(* Logix 5000 project; controller QA_DC vendor 1 type 14 code 164 rev 32.16; software revision 32.04 *)

TASK MainTask (continuous, watchdog 500 ms) : MainProgram, LN99, LN98

MODULES
   Local : vendor 1 type 14 code 164 (ICP 2, rev 32.16)
      QA_DC_ETHERNET : 1756-EN2T (ICP 1, Ethernet 10.28.22.45, rev 11.1)
         Schedule_PreProd : vendor 1 type 14 code 236 (Ethernet 10.28.22.40, rev 31.1, $0ec75abb$ RPI 20 ms, $0e455032$ RPI 20 ms, $6b8e262d$ RPI 20 ms, $a9dcfd1c$ RPI 20 ms, $64bd79af$ RPI 20 ms, $7c715bd6$ RPI 20 ms, $9c0a19c1$ RPI 20 ms, $e338eee0$ RPI 20 ms, $88140ee3$ RPI 20 ms, $4102ecba$ RPI 20 ms, $cc31c595$ RPI 20 ms, $3449dfe4$ RPI 20 ms, $565c2e57$ RPI 20 ms, $e38346de$ RPI 20 ms, $e483dda9$ RPI 20 ms, $e8d43428$ RPI 20 ms, $2ed72c0b$ RPI 20 ms, $3992ee42$ RPI 20 ms, $82c155fd$ RPI 20 ms, $a33d8fac$ RPI 20 ms)
END_MODULES

TYPE Barcode_SNModel :
STRUCT
   Data : STRING[5];
   Bit : BOOL[32];
END_STRUCT
END_TYPE

TYPE DateTime :
STRUCT
   Year : DINT;
   Month : DINT;
   Day : DINT;
   Hour : DINT;
   Minute : DINT;
   Seconds : DINT;
   Microseconds : DINT;
END_STRUCT
END_TYPE

TYPE DateTime_Type :   // Structure for the DateTime from the Controller wallclock accessed by the GSV/SSV instruction
STRUCT
   Year : DINT;
   Month : DINT;   // The month (1 - 12)
   Day : DINT;   // The day (1 - 31)
   Hour : DINT;   // hour (0 - 23)
   Minute : DINT;   // minute (0 - 59)
   Second : DINT;   // second (0 - 59)
   Microseconds : DINT;   // (0 - 999,999)
END_STRUCT
END_TYPE

TYPE STRING_12 :
STRUCT
   LEN : DINT;
   DATA : SINT[12];
END_STRUCT
END_TYPE

TYPE STRING_16 :
STRUCT
   LEN : DINT;
   DATA : SINT[16];
END_STRUCT
END_TYPE

TYPE STRING_24 :
STRUCT
   LEN : DINT;
   DATA : SINT[24];
END_STRUCT
END_TYPE

TYPE STRING_4 :
STRUCT
   LEN : DINT;
   DATA : SINT[4];
END_STRUCT
END_TYPE

TYPE STRING_40 :
STRUCT
   LEN : DINT;
   DATA : SINT[40];
END_STRUCT
END_TYPE

TYPE UDT_Current_Status :
STRUCT
   Area : STRING_12;
   Line : STRING_12;
   Shift : DINT;
   _1st_Shift_Avail : BOOL;
   _1st_Shift_Active : BOOL;
   _1st_Shift_Scheduled : BOOL;
   _2nd_Shift_Avail : BOOL;
   _2nd_Shift_Active : BOOL;
   _2nd_Shift_Scheduled : BOOL;
   _3rd_Shift_Avail : BOOL;
   _3rd_Shift_Active : BOOL;
   _3rd_Shift_Scheduled : BOOL;
   DayOfWeek : STRING_16;
   DayOfWeek_Int : DINT;
   Start_Time : STRING_16;
   End_Time : STRING_16;
   _1st_Break_Time : STRING_16;
   _1st_Break_Trigger : BOOL;
   _1st_Break_Active : BOOL;
   _1st_Break_Used : BOOL;
   Lunch_Time : STRING_16;
   Lunch_Trigger : BOOL;
   Lunch_Active : BOOL;
   Lunch_Used : BOOL;
   _2nd_Break_Time : STRING_16;
   _2nd_Break_Trigger : BOOL;
   _2nd_Break_Active : BOOL;
   _2nd_Break_Used : BOOL;
   Rotate_Active : BOOL;
   Rotate_Cmd : BOOL;   // 30 Second Downtime Event to Rotate the Crew
   Scheduled_Units : DINT;
   Line_Rate : DINT;   // Seconds to Construct a Component
   Line_Rate_SP : REAL;
   Units_Remaining : DINT;
   Units_Produced : DINT;
   Units_Scrapped : DINT;
   Units_Lossed : DINT;
   AY_Percent : REAL;
   Shift_Minutes_Remainng : DINT;
   Shift_Seconds_Remaining : DINT;
   DownTime_Code : DINT;
   Flex_Cmd : BOOL;
   Flex_Active : BOOL;
   FlexTo_Line : STRING_16;
   Flex_EndCmd : BOOL;
   Rotate_LEN : REAL;   // seconds
   Brk_LEN : REAL;   // minutes
   Lunch_LEN : REAL;   // minutes
   Break_Stop_On : BOOL;
   Break_Stop_Allowed : BOOL;
   Flex_Stop_On : BOOL;
   Flex_Stop_Allowed : BOOL;
   Rotate_Stop_On : BOOL;
   Rotate_Stop_Allowed : BOOL;
   S1_Scheduled : DINT;
   S2_Scheduled : DINT;
   S3_Scheduled : DINT;
   Shift_Scheduled : BOOL;
   Shift_Active : BOOL;
   RateToMakeSchedule : REAL;
   Theoretical_Units : DINT;
   Standard_LineRate : REAL;
   Running : BOOL;
   State : DINT;
   LineWide_Event : DINT;
   Units_Rejected : DINT;
END_STRUCT
END_TYPE

TYPE UDT_Daily_Schedule :
STRUCT
   _1st_Shift_Avail : BOOL;
   _1st_Shift_Start : STRING_16;
   _1st_Shift_End : STRING_16;
   _1st_Shift_Break1_Start : STRING_16;
   _1st_Shift_Break1_Length : DINT;   // Minutes
   _1st_Shift_Lunch_Start : STRING_16;
   _1st_Shift_Lunch_Length : DINT;   // Minutes
   _1st_Shift_Break2_Start : STRING_16;
   _1st_Shift_Break2_Length : DINT;   // Minutes
   _2nd_Shift_Avail : BOOL;
   _2nd_Shift_Start : STRING_16;
   _2nd_Shift_End : STRING_16;
   _2nd_Shift_Break1_Start : STRING_16;
   _2nd_Shift_Break1_Length : DINT;   // Minutes
   _2nd_Shift_Lunch_Start : STRING_16;
   _2nd_Shift_Lunch_Length : DINT;   // Minutes
   _2nd_Shift_Break2_Start : STRING_16;
   _2nd_Shift_Break2_Length : DINT;   // Minutes
   _3rd_Shift_Avail : BOOL;
   _3rd_Shift_Start : STRING_16;
   _3rd_Shift_End : STRING_16;
   _3rd_Shift_Break1_Start : STRING_16;
   _3rd_Shift_Break1_Length : DINT;   // Minutes
   _3rd_Shift_Lunch_Start : STRING_16;
   _3rd_Shift_Lunch_Length : DINT;   // Minutes
   _3rd_Shift_Break2_Start : STRING_16;
   _3rd_Shift_Break2_Length : DINT;   // Minutes
   Rotate_Length : DINT;   // Seconds
   Break_Stop_On : BOOL;
   Break_Stop_Allowed : BOOL;
   Flex_Stop_On : BOOL;
   Flex_Stop_Allowed : BOOL;
   Rotate_Stop_On : BOOL;
   Rotate_Stop_Allowed : BOOL;
   S1_Scheduled : DINT;
   S2_Scheduled : DINT;
   S3_Scheduled : DINT;
   RateToMakeSchedule : REAL;
END_STRUCT
END_TYPE

TYPE UDT_ShiftString_Breakdown :
STRUCT
   s1StartHour : STRING_4;
   s1StartMin : STRING_4;
   s1EndHour : STRING_4;
   s1_EndMin : STRING_4;
   s2StartHour : STRING_4;
   s2StartMin : STRING_4;
   s2EndHour : STRING_4;
   s2EndMin : STRING_4;
   s3StartHour : STRING_4;
   s3StartMin : STRING_4;
   s3EndHour : STRING_4;
   s3EndMin : STRING_4;
   break1StartHour : STRING_4;
   break1StartMin : STRING_4;
   break2StartHour : STRING_4;
   break2StartMin : STRING_4;
   lunchStartHour : STRING_4;
   lunchStartMin : STRING_4;
END_STRUCT
END_TYPE

TYPE UDT_SN_Model :
STRUCT
   writeIndex : DINT;
   readIndex : DINT;
   LastReadCode : DINT;
   Serial : STRING_16;
   Model : STRING_16;
   DateTime : STRING_24;
   newData : BOOL;
END_STRUCT
END_TYPE

TYPE UDT_Weekly_Schedule :
STRUCT
   Monday : UDT_Daily_Schedule;
   Tuesday : UDT_Daily_Schedule;
   Wednesday : UDT_Daily_Schedule;
   Thursday : UDT_Daily_Schedule;
   Friday : UDT_Daily_Schedule;
   Saturday : UDT_Daily_Schedule;
   Sunday : UDT_Daily_Schedule;
END_STRUCT
END_TYPE

VAR_GLOBAL   (* controller tags *)
   LN98_1st_Station_Break_Code : DINT;
   LN98_Break_LineWide : BOOL := 1;
   LN98_Current_Shift_Duration_Mins : DINT;
   LN98_Current_Shift_Duration_wBreaks_Mins : DINT := 510;
   LN98_DC_Controlled_Theoretical_Units : BOOL := 1;
   LN98_DT_CODE : DINT;
   LN98_FROM_DC1_MAIN_MESSAGES : DINT[20] := ([3] := 1000); {produced}
   LN98_NewDataModelSerial : BOOL;
   LN98_PreviousSerialNumber : STRING := 'XA1018189';
   LN98_Schedule : UDT_Current_Status := (DayOfWeek_Int := 4, Units_Produced := 1020, Theoretical_Units := 1000, LineWide_Event := 16, Units_Rejected := 34);
   LN98_Schedule_Cycle_Timer : TIMER := (PRE := 30600, ACC := 30400);
   LN98_Schedule_Max_Break_Duration : DINT := 60;
   LN98_Schedule_Max_Break_Timer : TIMER := (PRE := 3600000, ACC := 3600000, DN := 1);
   LN98_Schedule_TAKT : REAL := 30600.0;
   LN98_Scheduled_Units_Buffer : DINT := 1000;
   LN98_SerialNumber_ONS : BOOL;
   LN98_SerialNumberBuffer : STRING;
   LN98_SerialNumberChange_DelayTimer : TIMER := (PRE := 2000);
   LN98_SerialNumberChange_Timer : TIMER := (PRE := 3000);
   LN98_Shift_Reset_ONS : BOOL;
   LN98_Theoretical_Units_Counter : COUNTER := (PRE := 999999, ACC := 999);
   LN98_Theoretical_Units_Counter_ONS : BOOL;
   LN98_TO_DC01_DOWNTIME_CODE : DINT[10];   // DOWNTIME CODE CONSUME TAG
        [0]   // LN98
        [1]   // WORK CENTER MAIN LINE A
        [2]   // WORK CENTER MAIN LINE B
        [3]   // WORK CENTER MAIN LINE C
        [4]   // WORK CENTER MAIN LINE D
        [5]   // WORK CENTER MAIN LINE E
        [6]   // WORK CENTER SUB LINE C
        [7]   // WORK CENTER SUB LINE E
   LN98_TO_DC01_MAIN_MESSAGES : DINT[20] := ([4] := 1020, [16] := 34);   // KPI CONSUME TAG
        [17]   // ACTIVE SHIFT
        [18]   // SCHEDULED UNITS
        [19]   // LOST UNIT COUNT
        [4]   // ACTUAL UNIT COUNT
        [9]   // LINE STATUS
        [9].0   // LINE RUNNING
        [9].1   // LINE ON BREAK
        [9].2   // LINE ON FLEX STOP
   LN98_TO_DC01_MODEL_SERIAL_MESSAGE : STRING[2] := ([0] := 'WAXXXXXXXX 19', [1] := 'XA1018189');
   LN98_TO_DC1_MAIN_MESSAGE_A : DINT[10];   // WORK CENTER A CONSUME TAG
   LN98_TO_DC1_MAIN_MESSAGE_B : DINT[10];   // WORK CENTER B CONSUME TAG
   LN98_TO_DC1_MAIN_MESSAGE_C : DINT[10];   // WORK CENTER C CONSUME TAG
   LN98_TO_DC1_MAIN_MESSAGE_D : DINT[10];   // WORK CENTER D CONSUME TAG
   LN98_TO_DC1_MAIN_MESSAGE_E : DINT[10];   // WORK CENTER E CONSUME TAG
   LN98_TO_DC1_SUB_MESSAGE_C : DINT[10];   // WORK CENTER C CONSUME TAG
   LN98_TO_DC1_SUB_MESSAGE_E : DINT[10];   // WORK CENTER E CONSUME TAG
   LN98_Weekly_Schedule : UDT_Weekly_Schedule := (Monday._1st_Shift_Avail := 1, Monday._1st_Shift_Start := '2023-05-22 05:00', Monday._1st_Shift_End := '2023-05-22 14:30', Monday._2nd_Shift_Avail := 1, Monday._2nd_Shift_Start := '2023-05-22 16:45', Monday._2nd_Shift_End := '2023-05-23 03:15', Monday._3rd_Shift_Start := '2023-05-22 04:50', Monday._3rd_Shift_End := '2023-05-22 04:55', Monday.S1_Scheduled := 1000, Monday.S2_Scheduled := 1000, Tuesday._1st_Shift_Avail := 1, Tuesday._1st_Shift_Start := '2023-05-23 05:00', Tuesday._1st_Shift_End := '2023-05-23 14:30', Tuesday._2nd_Shift_Avail := 1, Tuesday._2nd_Shift_Start := '2023-05-23 16:45', Tuesday._2nd_Shift_End := '2023-05-24 03:15', Tuesday._3rd_Shift_Start := '2023-05-23 04:50', Tuesday._3rd_Shift_End := '2023-05-23 04:55', Tuesday.S1_Scheduled := 1000, Tuesday.S2_Scheduled := 1000, Wednesday._1st_Shift_Avail := 1, Wednesday._1st_Shift_Start := '2023-05-24 05:00', Wednesday._1st_Shift_End := '2023-05-24 14:30', Wednesday._2nd_Shift_Avail := 1, Wednesday._2nd_Shift_Start := '2023-05-24 16:45', Wednesday._2nd_Shift_End := '2023-05-25 03:15', Wednesday._3rd_Shift_Start := '2023-05-24 04:50', Wednesday._3rd_Shift_End := '2023-05-24 04:55', Wednesday.S1_Scheduled := 1000, Wednesday.S2_Scheduled := 1000, Thursday._1st_Shift_Avail := 1, Thursday._1st_Shift_Start := '2023-05-18 05:00', Thursday._1st_Shift_End := '2023-05-18 14:30', Thursday._2nd_Shift_Avail := 1, Thursday._2nd_Shift_Start := '2023-05-18 16:45', Thursday._2nd_Shift_End := '2023-05-19 03:15', Thursday._3rd_Shift_Start := '2023-05-18 04:50', Thursday._3rd_Shift_End := '2023-05-18 04:55', Thursday.S1_Scheduled := 1000, Thursday.S2_Scheduled := 1000, Friday._1st_Shift_Avail := 1, Friday._1st_Shift_Start := '2023-05-19 05:00', Friday._1st_Shift_End := '2023-05-19 14:30', Friday._2nd_Shift_Avail := 1, Friday._2nd_Shift_Start := '2023-05-19 16:45', Friday._2nd_Shift_End := '2023-05-20 03:15', Friday._3rd_Shift_Start := '2023-05-19 04:50', Friday._3rd_Shift_End := '2023-05-19 04:55', Friday.S1_Scheduled := 1000, Friday.S2_Scheduled := 1000, Saturday._1st_Shift_Start := '2023-05-20 05:00', Saturday._1st_Shift_End := '2023-05-20 14:30', Saturday._2nd_Shift_Start := '2023-05-20 16:45', Saturday._2nd_Shift_End := '2023-05-21 01:15', Saturday._3rd_Shift_Start := '2023-05-20 04:50', Saturday._3rd_Shift_End := '2023-05-20 04:55', Sunday._1st_Shift_Start := '2023-05-21 05:00', Sunday._1st_Shift_End := '2023-05-21 14:30', Sunday._2nd_Shift_Start := '2023-05-21 16:45', Sunday._2nd_Shift_End := '2023-05-22 01:15',
        Sunday._3rd_Shift_Start := '2023-05-21 04:50', Sunday._3rd_Shift_End := '2023-05-21 04:55');
   LN98_WORKCENTER_MAINLINE_A_DT_CODE : DINT;
   LN98_WORKCENTER_MAINLINE_B_DT_CODE : DINT;
   LN98_WORKCENTER_MAINLINE_C_DT_CODE : DINT;
   LN98_WORKCENTER_MAINLINE_D_DT_CODE : DINT;
   LN98_WORKCENTER_MAINLINE_E_DT_CODE : DINT;
   LN98_WORKCENTER_SUBLINE_C_DT_CODE : DINT;
   LN98_WORKCENTER_SUBLINE_E_DT_CODE : DINT;
   LN98ECS01 : DINT;
   LN98ECS02 : DINT;
   LN98ECS03 : DINT;
   LN98EES01 : DINT;
   LN98EES02 : DINT;
   LN98EES03 : DINT;
   LN98NAM01 : DINT;
   LN98NAM02 : DINT;
   LN98NAM03 : DINT;
   LN98NAM04 : DINT;
   LN98NBM01 : DINT;
   LN98NBM02 : DINT;
   LN98NBM03 : DINT;
   LN98NBM04 : DINT;
   LN98NCM01 : DINT;
   LN98NCM02 : DINT;
   LN98NCM04 : DINT;
   LN98NCM05 : DINT;
   LN98NDM01 : DINT;
   LN98NDM02 : DINT;
   LN98NDM03 : DINT;
   LN98NDM04 : DINT;
   LN98NEM01 : DINT;
   LN98NEM02 : DINT;
   LN98NEM03 : DINT;
   LN98NEM04 : DINT;
   LN98NEM05 : DINT;
   LN98SAM01 : DINT;
   LN98SAM02 : DINT;
   LN98SAM03 : DINT;
   LN98SAM04 : DINT;
   LN98SBM01 : DINT;
   LN98SBM02 : DINT;
   LN98SBM03 : DINT;
   LN98SBM04 : DINT;
   LN98SCM01 : DINT;
   LN98SCM02 : DINT;
   LN98SCM03 : DINT;
   LN98SCM04 : DINT;
   LN98SCM05 : DINT;
   LN98SDM01 : DINT;
   LN98SDM02 : DINT;
   LN98SDM03 : DINT;
   LN98SDM04 : DINT;
   LN98SEM01 : DINT;
   LN98SEM02 : DINT;
   LN98SEM04 : DINT;
   LN98SEM05 : DINT;
   LN98WCS01 : DINT;
   LN98WCS02 : DINT;
   LN98WCS03 : DINT;
   LN98WES01 : DINT;
   LN98WES02 : DINT;
   LN98WES03 : DINT;
   LN99_1st_Station_Break_Code : DINT;
   LN99_Break_LineWide : BOOL := 1;
   LN99_Current_Shift_Duration_Mins : DINT;
   LN99_Current_Shift_Duration_wBreaks_Mins : DINT := 460;
   LN99_DC_Controlled_Theoretical_Units : BOOL := 1;
   LN99_DT_CODE : DINT;
   LN99_FROM_DC1_MAIN_MESSAGES : DINT[20] := ([3] := 600); {produced}
   LN99_NewDataModelSerial : BOOL;
   LN99_PreviousSerialNumber : STRING := 'XB1017079';
   LN99_Schedule : UDT_Current_Status := (Line := 'LN01', _1st_Shift_Scheduled := 1, _2nd_Shift_Scheduled := 1, DayOfWeek := 'Tue', DayOfWeek_Int := 4, Start_Time := '2023-03-23 05:00', End_Time := '2023-03-23 14:30', Units_Remaining := 1452, Units_Produced := 766, Units_Lossed := 65, AY_Percent := 95.02853, Theoretical_Units := 1240, LineWide_Event := 16, Units_Rejected := 38);
   LN99_Schedule_Cycle_Timer : TIMER := (PRE := 22258, ACC := 2761);
   LN99_Schedule_Max_Break_Duration : DINT := 50;
   LN99_Schedule_Max_Break_Timer : TIMER := (PRE := 3000000, ACC := 2999998);
   LN99_Schedule_TAKT : REAL := 22258.064;
   LN99_Scheduled_Units_Buffer : DINT := 1240;
   LN99_SerialNumber_ONS : BOOL;
   LN99_SerialNumberBuffer : STRING;
   LN99_SerialNumberChange_DelayTimer : TIMER := (PRE := 2000);
   LN99_SerialNumberChange_Timer : TIMER := (PRE := 3000);
   LN99_Shift_Reset_ONS : BOOL;
   LN99_Theoretical_Units_Counter : COUNTER := (PRE := 999999, ACC := 1240);
   LN99_Theoretical_Units_Counter_ONS : BOOL;
   LN99_TO_DC01_DOWNTIME_CODE : DINT[10];   // DOWNTIME CODE CONSUME TAG
        [0]   // LN 99
        [1]   // WORK CENTER MAIN LINE A
        [2]   // WORK CENTER MAIN LINE B
        [3]   // WORK CENTER MAIN LINE C
        [4]   // WORK CENTER MAIN LINE D
        [5]   // WORK CENTER MAIN LINE E
        [6]   // WORK CENTER SUB LINE C
        [7]   // WORK CENTER SUB LINE E
   LN99_TO_DC01_MAIN_MESSAGES : DINT[20] := ([4] := 766, [16] := 38);   // KPI CONSUME TAG
        [17]   // ACTIVE SHIFT
        [18]   // SCHEDULED UNITS
        [19]   // LOST UNIT COUNT
        [4]   // ACTUAL UNIT COUNT
        [9]   // LINE STATUS
        [9].0   // LINE RUNNING
        [9].1   // LINE ON BREAK
        [9].2   // LINE ON FLEX STOP
   LN99_TO_DC01_MODEL_SERIAL_MESSAGE : STRING[2] := ([0] := 'WBXXXXXXXX 13', [1] := 'XB1017079');
   LN99_TO_DC1_MAIN_MESSAGE_A : DINT[10];   // WORK CENTER A CONSUME TAG
        [1]   // LN99NAM01
        [2]   // LN99SAM01
        [3]   // LN99NAM02
        [4]   // LN99SAM02
        [5]   // LN99NAM03
        [6]   // LN99SAM03
        [7]   // LN99NAM04
        [8]   // LN99SAM04
   LN99_TO_DC1_MAIN_MESSAGE_B : DINT[10];   // WORK CENTER B CONSUME TAG
        [1]   // LN99NBM01 WORK STATION
        [2]   // LN99SBM01 WORK STATION
        [3]   // LN99NBM02 WORK STATION
        [4]   // LN99SBM02 WORK STATION
        [5]   // LN99NBM03 WORK STATION
        [6]   // LN99SBM03 WORK STATION
        [7]   // LN99NBM04 WORK STATION
        [8]   // LN99SBM04 WORK STATION
   LN99_TO_DC1_MAIN_MESSAGE_C : DINT[10];   // WORK CENTER C CONSUME TAG
        [1]   // LN99NCM01 WORK STATION
        [2]   // LN99SCM01 WORK STATION
        [3]   // LN99NCM02 WORK STATION
        [4]   // LN99SCM02 WORK STATION
        [5]   // LN99SCM03 WORK STATION
        [6]   // LN99NCM04 WORK STATION
        [7]   // LN99SCM04 WORK STATION
        [8]   // LN99NCM05 WORK STATION
        [9]   // LN99SCM05 WORK STATION
   LN99_TO_DC1_MAIN_MESSAGE_D : DINT[10];   // WORK CENTER D CONSUME TAG
        [1]   // LN99NDM01 WORK STATION
        [2]   // LN99SDM01 WORK STATION
        [3]   // LN99NDM02 WORK STATION
        [4]   // LN99SDM02 WORK STATION
        [5]   // LN99NDM03 WORK STATION
        [6]   // LN99SDM03 WORK STATION
        [7]   // LN99NDM04 WORK STATION
        [8]   // LN99SDM04 WORK STATION
   LN99_TO_DC1_MAIN_MESSAGE_E : DINT[10];   // WORK CENTER E CONSUME TAG
        [1]   // LN99NEM01 WORK STATION
        [2]   // LN99SEM01 WORK STATION
        [3]   // LN99NEM02 WORK STATION
        [4]   // LN99SEM02 WORK STATION
        [5]   // LN99NEM03 WORK STATION
        [6]   // LN99NEM04 WORK STATION
        [7]   // LN99SEM04 WORK STATION
        [8]   // LN99NEM05 WORK STATION
        [9]   // LN99SEM05 WORK STATION
   LN99_TO_DC1_SUB_MESSAGE_C : DINT[10];   // WORK CENTER C CONSUME TAG
        [1]   // LN99WCS01 WORK STATION
        [2]   // LN99ECS01 WORK STATION
        [3]   // LN99WCS02 WORK STATION
        [4]   // LN99ECS02 WORK STATION
        [5]   // LN99WCS03 WORK STATION
        [6]   // LN99ECS03 WORK STATION
   LN99_TO_DC1_SUB_MESSAGE_E : DINT[10];   // WORK CENTER E CONSUME TAG
        [1]   // LN99WES01 WORK STATION
        [2]   // LN99EES01 WORK STATION
        [3]   // LN99WES02 WORK STATION
        [4]   // LN99EES02 WORK STATION
        [5]   // LN99WES03 WORK STATION
        [6]   // LN99EES03 WORK STATION
   LN99_Weekly_Schedule : UDT_Weekly_Schedule := (Monday._1st_Shift_Avail := 1, Monday._1st_Shift_Start := '2023-05-22 05:00', Monday._1st_Shift_End := '2023-05-22 13:30', Monday._2nd_Shift_Avail := 1, Monday._2nd_Shift_Start := '2023-05-22 16:45', Monday._2nd_Shift_End := '2023-05-23 01:15', Monday._3rd_Shift_Start := '2023-05-22 04:50', Monday._3rd_Shift_End := '2023-05-22 04:55', Monday.S1_Scheduled := 1240, Monday.S2_Scheduled := 1240, Tuesday._1st_Shift_Avail := 1, Tuesday._1st_Shift_Start := '2023-05-23 05:00', Tuesday._1st_Shift_End := '2023-05-23 13:30', Tuesday._2nd_Shift_Avail := 1, Tuesday._2nd_Shift_Start := '2023-05-23 16:45', Tuesday._2nd_Shift_End := '2023-05-24 01:15', Tuesday._3rd_Shift_Start := '2023-05-23 04:50', Tuesday._3rd_Shift_End := '2023-05-23 04:55', Tuesday.S1_Scheduled := 1240, Tuesday.S2_Scheduled := 1240, Wednesday._1st_Shift_Avail := 1, Wednesday._1st_Shift_Start := '2023-05-24 05:00', Wednesday._1st_Shift_End := '2023-05-24 13:30', Wednesday._2nd_Shift_Avail := 1, Wednesday._2nd_Shift_Start := '2023-05-24 16:45', Wednesday._2nd_Shift_End := '2023-05-25 01:15', Wednesday._3rd_Shift_Start := '2023-05-24 04:50', Wednesday._3rd_Shift_End := '2023-05-24 04:55', Wednesday.S1_Scheduled := 1240, Wednesday.S2_Scheduled := 1240, Thursday._1st_Shift_Avail := 1, Thursday._1st_Shift_Start := '2023-05-18 05:00', Thursday._1st_Shift_End := '2023-05-18 13:30', Thursday._2nd_Shift_Avail := 1, Thursday._2nd_Shift_Start := '2023-05-18 16:45', Thursday._2nd_Shift_End := '2023-05-19 01:15', Thursday._3rd_Shift_Start := '2023-05-18 04:50', Thursday._3rd_Shift_End := '2023-05-18 04:55', Thursday.S1_Scheduled := 1240, Thursday.S2_Scheduled := 1240, Friday._1st_Shift_Avail := 1, Friday._1st_Shift_Start := '2023-05-19 05:00', Friday._1st_Shift_End := '2023-05-19 13:30', Friday._2nd_Shift_Avail := 1, Friday._2nd_Shift_Start := '2023-05-19 16:45', Friday._2nd_Shift_End := '2023-05-20 01:15', Friday._3rd_Shift_Start := '2023-05-19 04:50', Friday._3rd_Shift_End := '2023-05-19 04:55', Friday.S1_Scheduled := 1240, Friday.S2_Scheduled := 1240, Saturday._1st_Shift_Start := '2023-05-20 05:00', Saturday._1st_Shift_End := '2023-05-20 13:30', Saturday._2nd_Shift_Start := '2023-05-20 16:45', Saturday._2nd_Shift_End := '2023-05-21 01:15', Saturday._3rd_Shift_Start := '2023-05-20 04:50', Saturday._3rd_Shift_End := '2023-05-20 04:55', Saturday.S1_Scheduled := 1240, Saturday.S2_Scheduled := 1240, Sunday._1st_Shift_Start := '2023-05-21 05:00', Sunday._1st_Shift_End := '2023-05-21 13:30',
        Sunday._2nd_Shift_Start := '2023-05-21 16:45', Sunday._2nd_Shift_End := '2023-05-22 01:15', Sunday._3rd_Shift_Start := '2023-05-21 04:50', Sunday._3rd_Shift_End := '2023-05-21 04:55', Sunday.S1_Scheduled := 1240, Sunday.S2_Scheduled := 1240);
   LN99_WORKCENTER_MAINLINE_A_DT_CODE : DINT;
   LN99_WORKCENTER_MAINLINE_B_DT_CODE : DINT;
   LN99_WORKCENTER_MAINLINE_C_DT_CODE : DINT;
   LN99_WORKCENTER_MAINLINE_D_DT_CODE : DINT;
   LN99_WORKCENTER_MAINLINE_E_DT_CODE : DINT;
   LN99_WORKCENTER_SUBLINE_C_DT_CODE : DINT;
   LN99_WORKCENTER_SUBLINE_E_DT_CODE : DINT;
   LN99ECS01 : DINT;   // WORK STATION EAST SIDE WORKCENTER C SUBLINE STATION 01
   LN99ECS02 : DINT;   // WORK STATION EAST SIDE WORKCENTER C SUBLINE STATION 02
   LN99ECS03 : DINT;   // WORK STATION EAST SIDE WORKCENTER C SUBLINE STATION 03
   LN99EES01 : DINT;   // WORK STATION EAST SIDE WORK CENTER E SUBLINE STATION 01
   LN99EES02 : DINT;   // WORK STATION EAST SIDE WORK CENTER E SUBLINE STATION 02
   LN99EES03 : DINT;   // WORK STATION EAST SIDE WORK CENTER E SUBLINE STATION 03
   LN99NAM01 : DINT;   // WORKSTATION NORTH SIDE WORKCENTER A MAIN LINE STATION 01
   LN99NAM02 : DINT;   // WORKSTATION NORTH SIDE WORKCENTER A MAINLINE STATION 02
   LN99NAM03 : DINT;   // WORKSTATION NORTH SIDE WORKCENTER A MAINLINE STATION 03
   LN99NAM04 : DINT;   // WORKSTATION NORTH SIDE WORKCENTER A MAINLINE STATION 04
   LN99NBM01 : DINT;   // WORK STATION NORTH SIDE WORKCENTER B MAINLINE STATION 01
   LN99NBM02 : DINT;   // WORK STATION NORTH SIDE WORKCENTER B MAINLINE STATION 02
   LN99NBM03 : DINT;   // WORK STATION NORTH SIDE WORKCENTER B MAINLINE STATION 03
   LN99NBM04 : DINT;   // WORK STATION NORTH SIDE WORKCENTER B MAINLINE STATION 4
   LN99NCM01 : DINT;   // WORK STATION NORTH SIDE WORKCENTER C MAINLINE STATION 01
   LN99NCM02 : DINT;   // WORK STATION NORTH SIDE WORKCENTER C MAINLINE STATION 02
   LN99NCM04 : DINT;   // WORK STATION NORTH SIDE WORKCENTER C MAINLINE STATION 04
   LN99NCM05 : DINT;   // WORK STATION NORTH SIDE WORKCENTER C MAINLINE STATION 05
   LN99NDM01 : DINT;   // WORK STATION NORTH SIDE WORKCENTER D MAINLINE STATION 01
   LN99NDM02 : DINT;   // WORK STATION NORTH SIDE WORK CENTER D MAINLINE STATION 02
   LN99NDM03 : DINT;   // WORK STATION NORTH SIDE WORK CENTER D MAINLINE STATION 03
   LN99NDM04 : DINT;   // WORK STATION NORTH SIDE WORK CENTER D MAINLINE STATION 04
   LN99NEM01 : DINT;   // WORK STATION NORTH SIDE WORK CENTER E MAIN LINE STATION 01
   LN99NEM02 : DINT;   // WORK STATION NORTH SIDE WORK CENTER E MAINLINE STATION 02
   LN99NEM03 : DINT;   // WORK STATION NORTH SIDE WORK CENTER E MAINLINE STATION 03
   LN99NEM04 : DINT;   // WORK STATION NORTH SIDE WORK CENTER E MAINLINE STATION 04
   LN99NEM05 : DINT;   // WORK STATION NORTH SIDE WORK CENTER E MAINLINE STATION 05
   LN99SAM01 : DINT;   // WORKSTATION SOUTH SIDE WORKCENTER A MAIN LINE STATION 01
   LN99SAM02 : DINT;   // WORKSTATION SOUTH SIDE WORKCENTER A MAINLINE STATION 02
   LN99SAM03 : DINT;   // WORKSTATION SOUTH SIDE WORKCENTER A MAINLINE STATION 03
   LN99SAM04 : DINT;   // WORKSTATION SOUTH SIDE WORKCENTER A MAINLINE STATION 04
   LN99SBM01 : DINT;   // WORK STATION SOUTH SIDE WORKCENTER B MAINLINE STATION 01
   LN99SBM02 : DINT;   // WORK STATION SOUTH SIDE WORKCENTER B MAINLINE STATION 02
   LN99SBM03 : DINT;   // WORK STATION SOUTH SIDE WORKCENTER B MAINLINE STATION 03
   LN99SBM04 : DINT;   // WORK STATION SOUTH SIDE WORKCENTER B MAINLINE STATION 04
   LN99SCM01 : DINT;   // WORK STATION SOUTH SIDE WORKCENTER C MAINLINE STATION 01
   LN99SCM02 : DINT;   // WORK STATION SOUTH SIDE WORKCENTER C MAINLINE STATION 02
   LN99SCM03 : DINT;   // WORK STATION SOUTH SIDE WORKCENTER C MAINLINE STATION 03
   LN99SCM04 : DINT;   // WORK STATION SOUTH SIDE WORKCENTER C MAINLINE STATION 04
   LN99SCM05 : DINT;   // WORK STATION SOUTH SIDE WORKCENTER C MAINLINE STATION 05
   LN99SDM01 : DINT;   // WORK STATION SOUTH SIDE WORKCENTER D MAINLINE STATION 01
   LN99SDM02 : DINT;   // WORK STATION SOUTH SIDE WORK CENTER D MAINLINE STATION 02
   LN99SDM03 : DINT;   // WORK STATION SOUTH SIDE WORK CENTER D MAINLINE STATION 03
   LN99SDM04 : DINT;   // WORK STATION SOUTH SIDE WORK CENTER D MAINLINE STATION 04
   LN99SEM01 : DINT;   // WORK STATION SOUTH SIDE WORK CENTER E MAINLINE STATION 01
   LN99SEM02 : DINT;   // WORK STATION SOUTH SIDE WORK CENTER E MAINLINE STATION 02
   LN99SEM04 : DINT;   // WORK STATION SOUTH SIDE WORK CENTER E MAINLINE STATION 04
   LN99SEM05 : DINT;   // WORK STATION SOUTH SIDE WORK CENTER E MAINLINE STATION 05
   LN99WCS01 : DINT;   // WORK STATION WEST SIDE WORKCENTER C SUBLINE STATION 01
   LN99WCS02 : DINT;   // WORK STATION WEST SIDE WORKCENTER C SUBLINE STATION 02
   LN99WCS03 : DINT;   // WORK STATION WEST SIDE WORKCENTER C SUBLINE STATION 03
   LN99WES01 : DINT;   // WORK STATION WEST SIDE WORK CENTER E SUBLINE STATION 01
   LN99WES02 : DINT;   // WORK STATION WEST SIDE WORK CENTER E SUBLINE STATION 02
   LN99WES03 : DINT;   // WORK STATION WEST SIDE WORK CENTER E SUBLINE STATION 03
END_VAR

PROGRAM LN98   (* main routine MainRoutine *)

ROUTINE MainRoutine   (* ladder *)
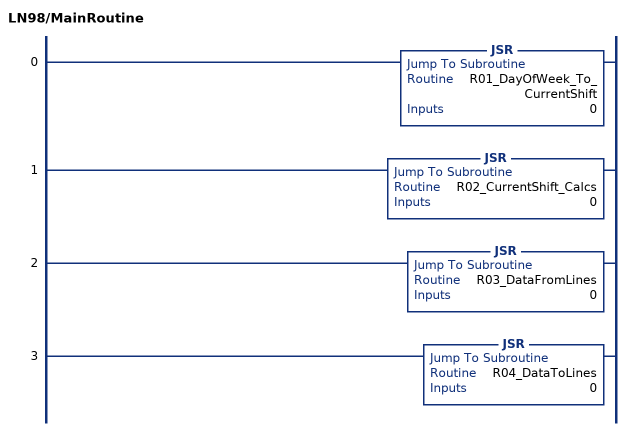
   0: JSR(R01_DayOfWeek_To_CurrentShift,0);
   1: JSR(R02_CurrentShift_Calcs,0);
   2: JSR(R03_DataFromLines,0);
   3: JSR(R04_DataToLines,0);
END_ROUTINE

ROUTINE R01_DayOfWeek_To_CurrentShift   (* ladder *)
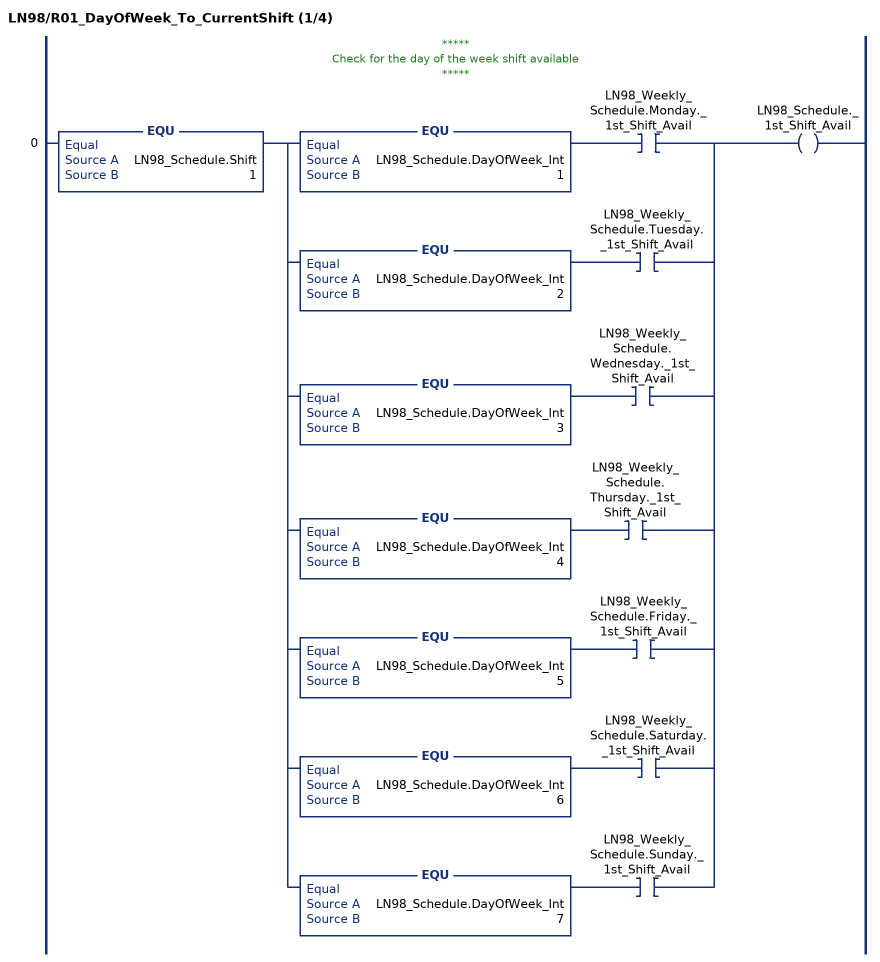
   // *****
   // Check for the day of the week shift available
   // *****
   0: EQU(LN98_Schedule.Shift,1)[EQU(LN98_Schedule.DayOfWeek_Int,1) XIC(LN98_Weekly_Schedule.Monday._1st_Shift_Avail) ,EQU(LN98_Schedule.DayOfWeek_Int,2) XIC(LN98_Weekly_Schedule.Tuesday._1st_Shift_Avail) ,EQU(LN98_Schedule.DayOfWeek_Int,3) XIC(LN98_Weekly_Schedule.Wednesday._1st_Shift_Avail) ,EQU(LN98_Schedule.DayOfWeek_Int,4) XIC(LN98_Weekly_Schedule.Thursday._1st_Shift_Avail) ,EQU(LN98_Schedule.DayOfWeek_Int,5) XIC(LN98_Weekly_Schedule.Friday._1st_Shift_Avail) ,EQU(LN98_Schedule.DayOfWeek_Int,6) XIC(LN98_Weekly_Schedule.Saturday._1st_Shift_Avail) ,EQU(LN98_Schedule.DayOfWeek_Int,7) XIC(LN98_Weekly_Schedule.Sunday._1st_Shift_Avail) ]OTE(LN98_Schedule._1st_Shift_Avail);
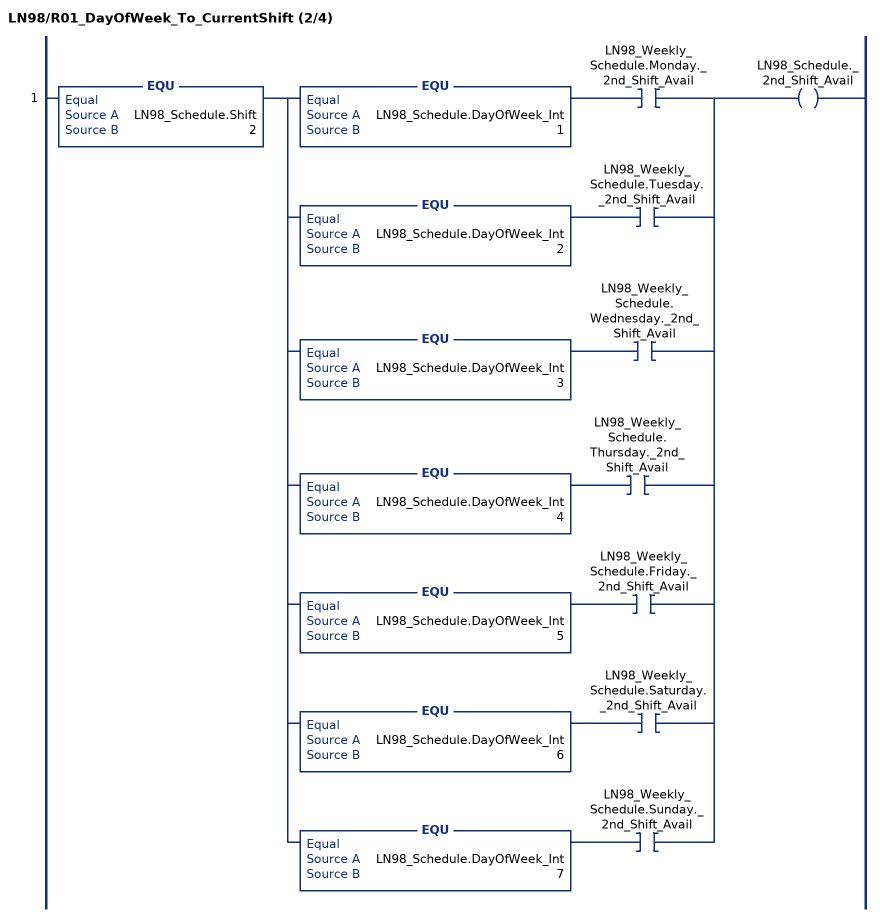
   1: EQU(LN98_Schedule.Shift,2)[EQU(LN98_Schedule.DayOfWeek_Int,1) XIC(LN98_Weekly_Schedule.Monday._2nd_Shift_Avail) ,EQU(LN98_Schedule.DayOfWeek_Int,2) XIC(LN98_Weekly_Schedule.Tuesday._2nd_Shift_Avail) ,EQU(LN98_Schedule.DayOfWeek_Int,3) XIC(LN98_Weekly_Schedule.Wednesday._2nd_Shift_Avail) ,EQU(LN98_Schedule.DayOfWeek_Int,4) XIC(LN98_Weekly_Schedule.Thursday._2nd_Shift_Avail) ,EQU(LN98_Schedule.DayOfWeek_Int,5) XIC(LN98_Weekly_Schedule.Friday._2nd_Shift_Avail) ,EQU(LN98_Schedule.DayOfWeek_Int,6) XIC(LN98_Weekly_Schedule.Saturday._2nd_Shift_Avail) ,EQU(LN98_Schedule.DayOfWeek_Int,7) XIC(LN98_Weekly_Schedule.Sunday._2nd_Shift_Avail) ]OTE(LN98_Schedule._2nd_Shift_Avail);
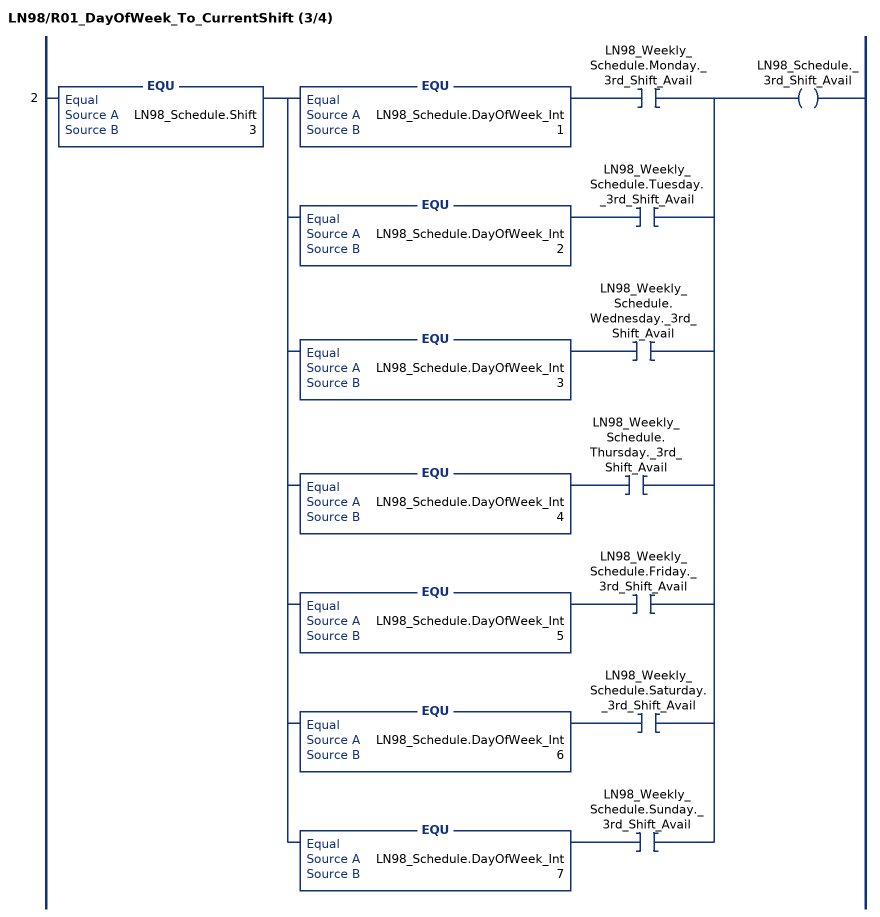
   2: EQU(LN98_Schedule.Shift,3)[EQU(LN98_Schedule.DayOfWeek_Int,1) XIC(LN98_Weekly_Schedule.Monday._3rd_Shift_Avail) ,EQU(LN98_Schedule.DayOfWeek_Int,2) XIC(LN98_Weekly_Schedule.Tuesday._3rd_Shift_Avail) ,EQU(LN98_Schedule.DayOfWeek_Int,3) XIC(LN98_Weekly_Schedule.Wednesday._3rd_Shift_Avail) ,EQU(LN98_Schedule.DayOfWeek_Int,4) XIC(LN98_Weekly_Schedule.Thursday._3rd_Shift_Avail) ,EQU(LN98_Schedule.DayOfWeek_Int,5) XIC(LN98_Weekly_Schedule.Friday._3rd_Shift_Avail) ,EQU(LN98_Schedule.DayOfWeek_Int,6) XIC(LN98_Weekly_Schedule.Saturday._3rd_Shift_Avail) ,EQU(LN98_Schedule.DayOfWeek_Int,7) XIC(LN98_Weekly_Schedule.Sunday._3rd_Shift_Avail) ]OTE(LN98_Schedule._3rd_Shift_Avail);
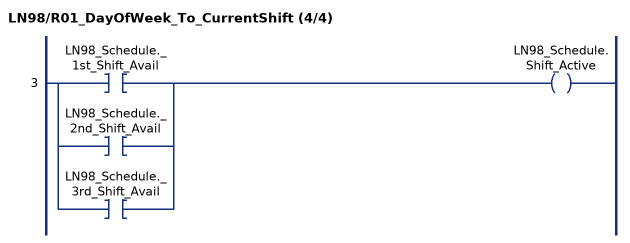
   3: [XIC(LN98_Schedule._1st_Shift_Avail) ,XIC(LN98_Schedule._2nd_Shift_Avail) ,XIC(LN98_Schedule._3rd_Shift_Avail) ]OTE(LN98_Schedule.Shift_Active);
END_ROUTINE

ROUTINE R02_CurrentShift_Calcs   (* ladder *)
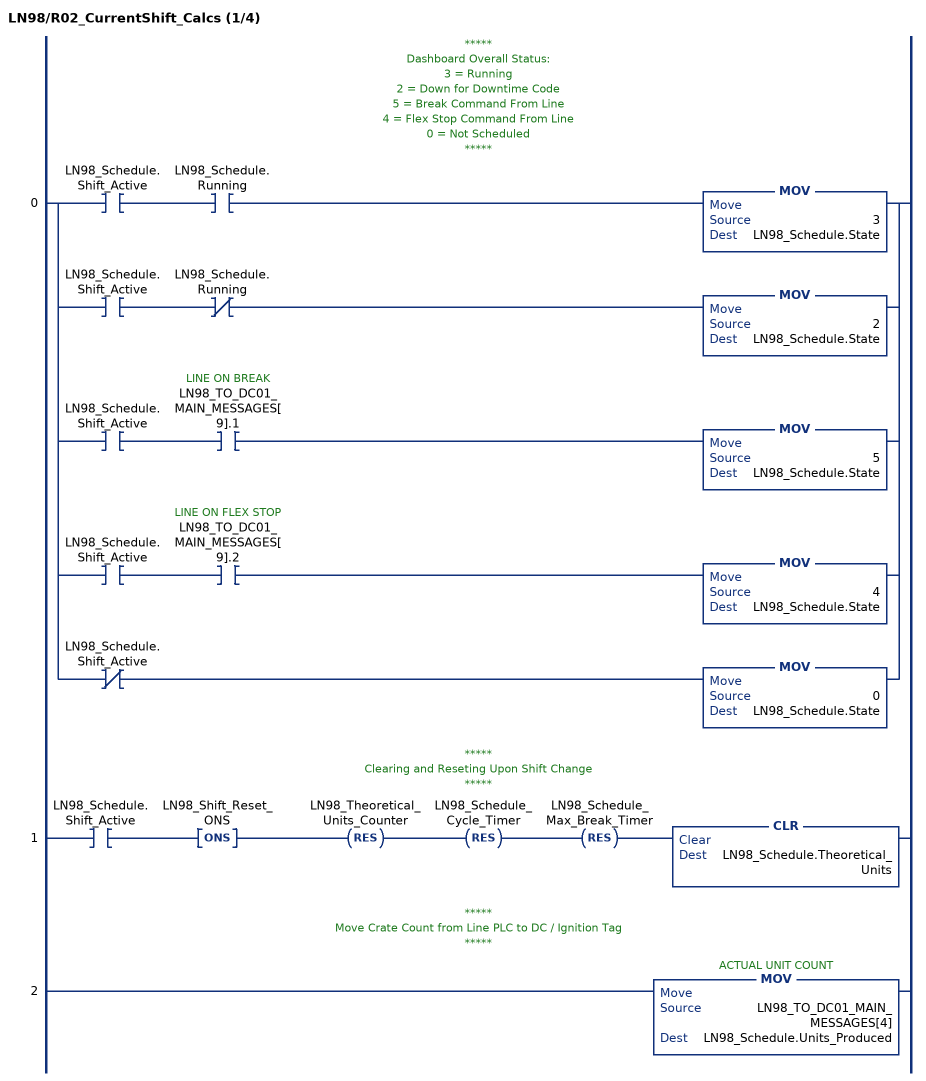
   // *****
   // Dashboard Overall Status:
   // 3 = Running
   // 2 = Down for Downtime Code
   // 5 = Break Command From Line
   // 4 = Flex Stop Command From Line
   // 0 = Not Scheduled
   // *****
   0: [XIC(LN98_Schedule.Shift_Active) XIC(LN98_Schedule.Running) MOV(3,LN98_Schedule.State) ,XIC(LN98_Schedule.Shift_Active) XIO(LN98_Schedule.Running) MOV(2,LN98_Schedule.State) ,XIC(LN98_Schedule.Shift_Active) XIC(LN98_TO_DC01_MAIN_MESSAGES[9].1) MOV(5,LN98_Schedule.State) ,XIC(LN98_Schedule.Shift_Active) XIC(LN98_TO_DC01_MAIN_MESSAGES[9].2) MOV(4,LN98_Schedule.State) ,XIO(LN98_Schedule.Shift_Active) MOV(0,LN98_Schedule.State) ];
   // *****
   // Clearing and Reseting Upon Shift Change
   // *****
   1: XIC(LN98_Schedule.Shift_Active)ONS(LN98_Shift_Reset_ONS)RES(LN98_Theoretical_Units_Counter)RES(LN98_Schedule_Cycle_Timer)RES(LN98_Schedule_Max_Break_Timer)CLR(LN98_Schedule.Theoretical_Units);
   // *****
   // Move Crate Count from Line PLC to DC / Ignition Tag
   // *****
   2: MOV(LN98_TO_DC01_MAIN_MESSAGES[4],LN98_Schedule.Units_Produced);
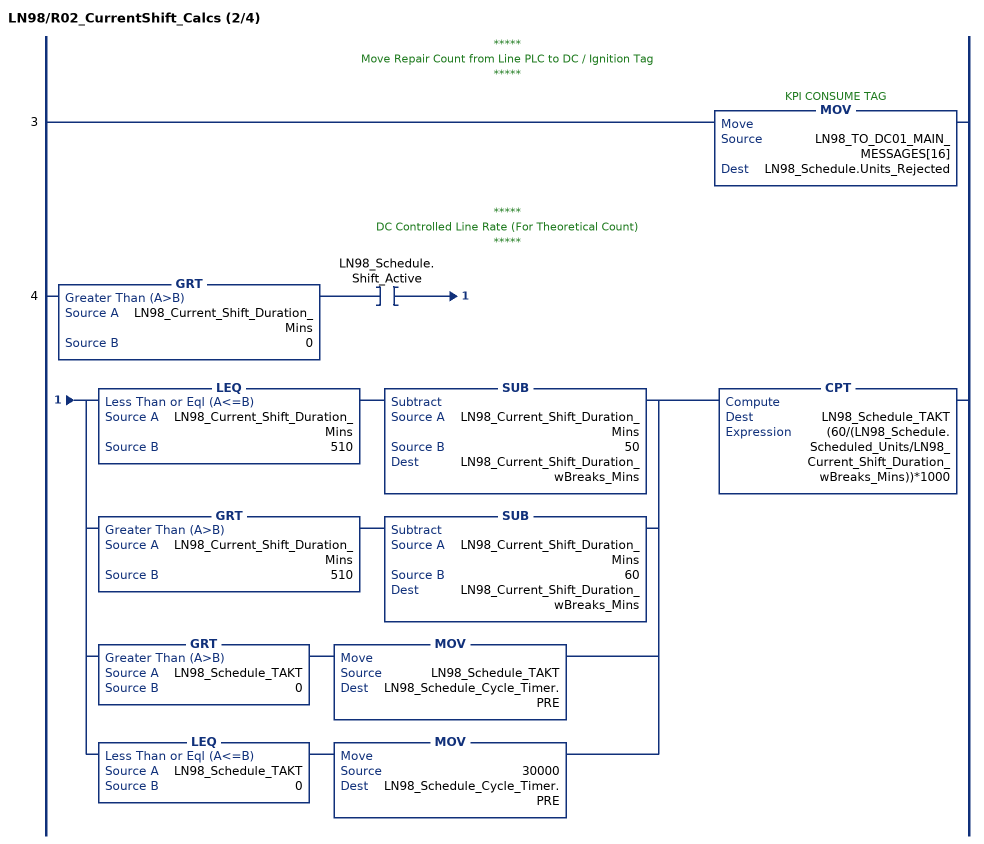
   // *****
   // Move Repair Count from Line PLC to DC / Ignition Tag
   // *****
   3: MOV(LN98_TO_DC01_MAIN_MESSAGES[16],LN98_Schedule.Units_Rejected);
   // *****
   // DC Controlled Line Rate (For Theoretical Count)
   // *****
   4: GRT(LN98_Current_Shift_Duration_Mins,0)XIC(LN98_Schedule.Shift_Active)[LEQ(LN98_Current_Shift_Duration_Mins,510) SUB(LN98_Current_Shift_Duration_Mins,50,LN98_Current_Shift_Duration_wBreaks_Mins) ,GRT(LN98_Current_Shift_Duration_Mins,510) SUB(LN98_Current_Shift_Duration_Mins,60,LN98_Current_Shift_Duration_wBreaks_Mins) ,GRT(LN98_Schedule_TAKT,0) MOV(LN98_Schedule_TAKT,LN98_Schedule_Cycle_Timer.PRE) ,LEQ(LN98_Schedule_TAKT,0) MOV(30000,LN98_Schedule_Cycle_Timer.PRE) ]CPT(LN98_Schedule_TAKT,(60/(LN98_Schedule.Scheduled_Units/LN98_Current_Shift_Duration_wBreaks_Mins))*1000);
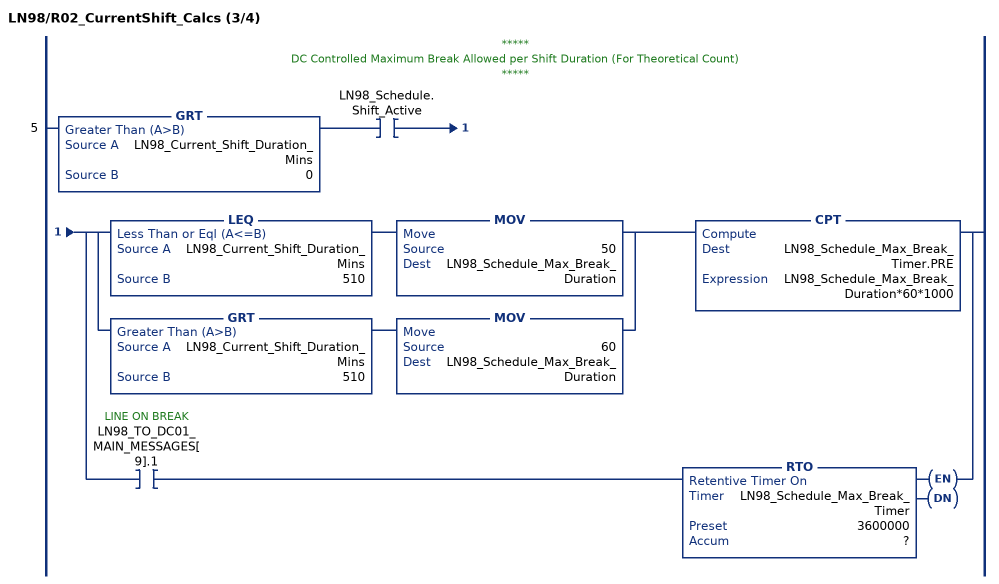
   // *****
   // DC Controlled Maximum Break Allowed per Shift Duration (For Theoretical Count)
   // *****
   5: GRT(LN98_Current_Shift_Duration_Mins,0)XIC(LN98_Schedule.Shift_Active)[[LEQ(LN98_Current_Shift_Duration_Mins,510) MOV(50,LN98_Schedule_Max_Break_Duration) ,GRT(LN98_Current_Shift_Duration_Mins,510) MOV(60,LN98_Schedule_Max_Break_Duration) ] CPT(LN98_Schedule_Max_Break_Timer.PRE,LN98_Schedule_Max_Break_Duration*60*1000) ,XIC(LN98_TO_DC01_MAIN_MESSAGES[9].1) RTO(LN98_Schedule_Max_Break_Timer,?,?) ];
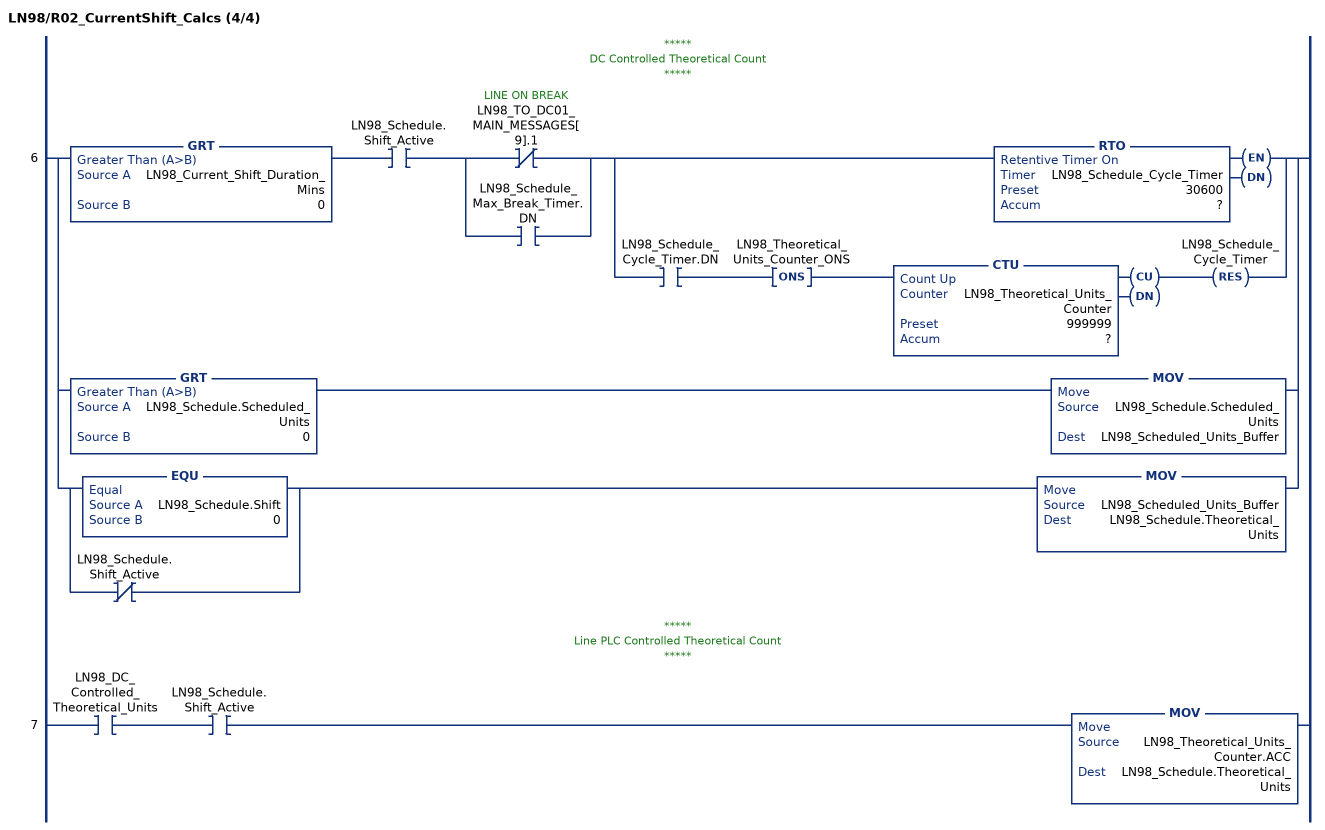
   // *****
   // DC Controlled Theoretical Count
   // *****
   6: [GRT(LN98_Current_Shift_Duration_Mins,0) XIC(LN98_Schedule.Shift_Active) [XIO(LN98_TO_DC01_MAIN_MESSAGES[9].1) ,XIC(LN98_Schedule_Max_Break_Timer.DN) ] [RTO(LN98_Schedule_Cycle_Timer,?,?) ,XIC(LN98_Schedule_Cycle_Timer.DN) ONS(LN98_Theoretical_Units_Counter_ONS) CTU(LN98_Theoretical_Units_Counter,?,?) RES(LN98_Schedule_Cycle_Timer) ] ,GRT(LN98_Schedule.Scheduled_Units,0) MOV(LN98_Schedule.Scheduled_Units,LN98_Scheduled_Units_Buffer) ,[EQU(LN98_Schedule.Shift,0) ,XIO(LN98_Schedule.Shift_Active) ] MOV(LN98_Scheduled_Units_Buffer,LN98_Schedule.Theoretical_Units) ];
   // *****
   // Line PLC Controlled Theoretical Count
   // *****
   7: XIC(LN98_DC_Controlled_Theoretical_Units)XIC(LN98_Schedule.Shift_Active)MOV(LN98_Theoretical_Units_Counter.ACC,LN98_Schedule.Theoretical_Units);
END_ROUTINE

ROUTINE R03_DataFromLines   (* ladder *)
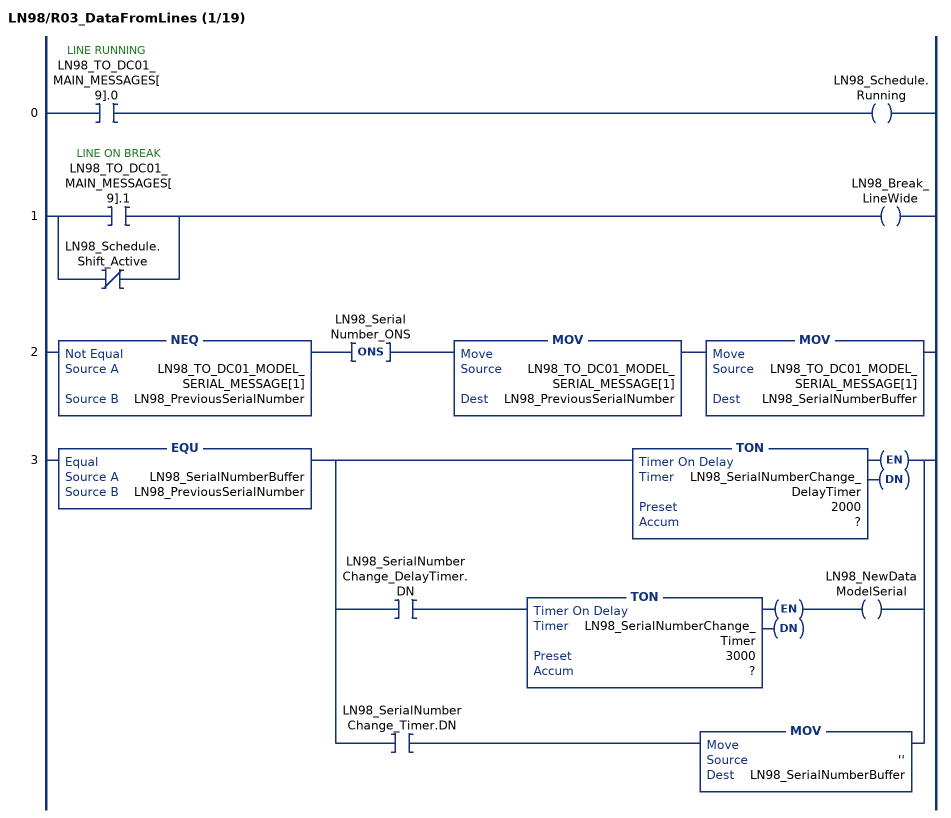
   0: XIC(LN98_TO_DC01_MAIN_MESSAGES[9].0)OTE(LN98_Schedule.Running);
   1: [XIC(LN98_TO_DC01_MAIN_MESSAGES[9].1) ,XIO(LN98_Schedule.Shift_Active) ]OTE(LN98_Break_LineWide);
   2: NEQ(LN98_TO_DC01_MODEL_SERIAL_MESSAGE[1],LN98_PreviousSerialNumber)ONS(LN98_SerialNumber_ONS)MOV(LN98_TO_DC01_MODEL_SERIAL_MESSAGE[1],LN98_PreviousSerialNumber)MOV(LN98_TO_DC01_MODEL_SERIAL_MESSAGE[1],LN98_SerialNumberBuffer);
   3: EQU(LN98_SerialNumberBuffer,LN98_PreviousSerialNumber)[TON(LN98_SerialNumberChange_DelayTimer,?,?) ,XIC(LN98_SerialNumberChange_DelayTimer.DN) TON(LN98_SerialNumberChange_Timer,?,?) OTE(LN98_NewDataModelSerial) ,XIC(LN98_SerialNumberChange_Timer.DN) MOV('',LN98_SerialNumberBuffer) ];
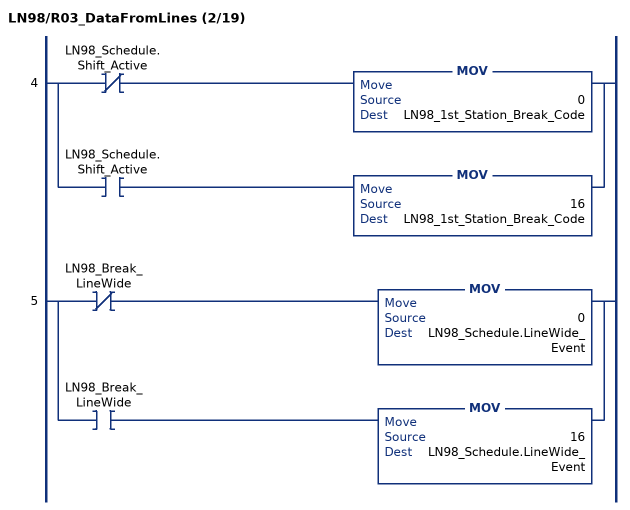
   4: [XIO(LN98_Schedule.Shift_Active) MOV(0,LN98_1st_Station_Break_Code) ,XIC(LN98_Schedule.Shift_Active) MOV(16,LN98_1st_Station_Break_Code) ];
   5: [XIO(LN98_Break_LineWide) MOV(0,LN98_Schedule.LineWide_Event) ,XIC(LN98_Break_LineWide) MOV(16,LN98_Schedule.LineWide_Event) ];
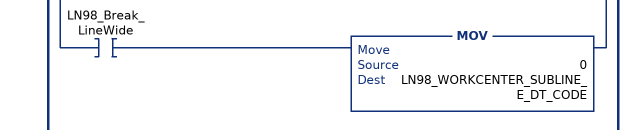
   // MNT Faults
   // If an MNT workcenter is tied to the main line or subline where there is already a workcenter with a workstaiton where "LN98_Break_LineWide (when high) MOVEs a 16 in, then that MNT can MOVE a 0 in when "LN98_Break_LineWide" goes high
   // If it is an independent MNT (not tied to a workcenter), "LN98_Break_LineWide" Tag should MOVE a 16 when "LN98_Break_LineWide" goes high
   6: [XIO(LN98_Break_LineWide) MOV(LN98_TO_DC01_DOWNTIME_CODE[0],LN98_DT_CODE) ,XIC(LN98_Break_LineWide) MOV(0,LN98_DT_CODE) ,XIO(LN98_Break_LineWide) MOV(LN98_TO_DC01_DOWNTIME_CODE[1],LN98_WORKCENTER_MAINLINE_A_DT_CODE) ,XIC(LN98_Break_LineWide) MOV(0,LN98_WORKCENTER_MAINLINE_A_DT_CODE) ,XIO(LN98_Break_LineWide) MOV(LN98_TO_DC01_DOWNTIME_CODE[2],LN98_WORKCENTER_MAINLINE_B_DT_CODE) ,XIC(LN98_Break_LineWide) MOV(0,LN98_WORKCENTER_MAINLINE_B_DT_CODE) ,XIO(LN98_Break_LineWide) MOV(LN98_TO_DC01_DOWNTIME_CODE[3],LN98_WORKCENTER_MAINLINE_C_DT_CODE) ,XIC(LN98_Break_LineWide) MOV(0,LN98_WORKCENTER_MAINLINE_C_DT_CODE) ,XIO(LN98_Break_LineWide) MOV(LN98_TO_DC01_DOWNTIME_CODE[4],LN98_WORKCENTER_MAINLINE_D_DT_CODE) ,XIC(LN98_Break_LineWide) MOV(0,LN98_WORKCENTER_MAINLINE_D_DT_CODE) ,XIO(LN98_Break_LineWide) MOV(LN98_TO_DC01_DOWNTIME_CODE[5],LN98_WORKCENTER_MAINLINE_E_DT_CODE) ,XIC(LN98_Break_LineWide) MOV(0,LN98_WORKCENTER_MAINLINE_E_DT_CODE) ,XIO(LN98_Break_LineWide) MOV(LN98_TO_DC01_DOWNTIME_CODE[6],LN98_WORKCENTER_SUBLINE_C_DT_CODE) ,XIC(LN98_Break_LineWide) MOV(0,LN98_WORKCENTER_SUBLINE_C_DT_CODE) ,XIO(LN98_Break_LineWide) MOV(LN98_TO_DC01_DOWNTIME_CODE[7],LN98_WORKCENTER_SUBLINE_E_DT_CODE) ,XIC(LN98_Break_LineWide) MOV(0,LN98_WORKCENTER_SUBLINE_E_DT_CODE) ];
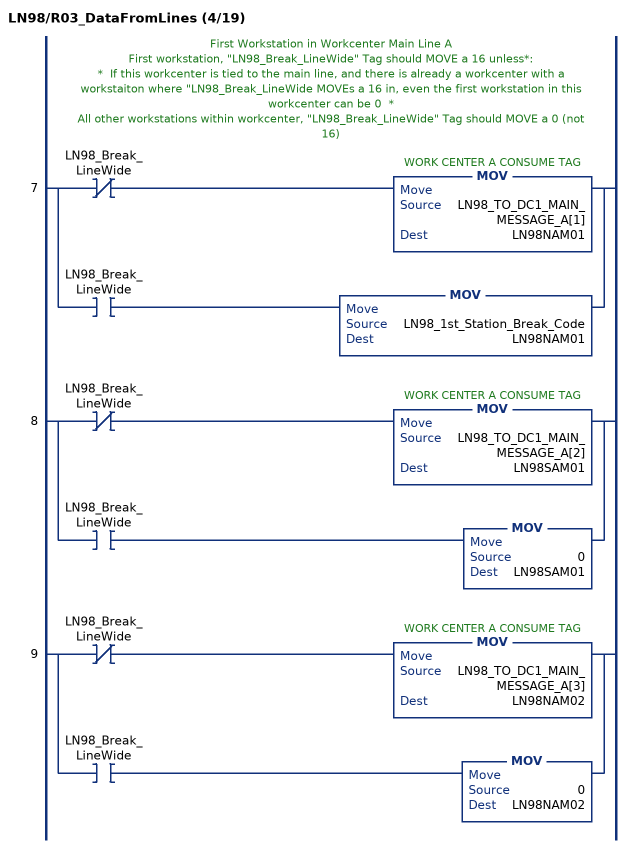
   // First Workstation in Workcenter Main Line A
   // First workstation, "LN98_Break_LineWide" Tag should MOVE a 16 unless*:
   // *  If this workcenter is tied to the main line, and there is already a workcenter with a workstaiton where "LN98_Break_LineWide MOVEs a 16 in, even the first workstation in this workcenter can be 0  *
   // All other workstations within workcenter, "LN98_Break_LineWide" Tag should MOVE a 0 (not 16)
   7: [XIO(LN98_Break_LineWide) MOV(LN98_TO_DC1_MAIN_MESSAGE_A[1],LN98NAM01) ,XIC(LN98_Break_LineWide) MOV(LN98_1st_Station_Break_Code,LN98NAM01) ];
   8: [XIO(LN98_Break_LineWide) MOV(LN98_TO_DC1_MAIN_MESSAGE_A[2],LN98SAM01) ,XIC(LN98_Break_LineWide) MOV(0,LN98SAM01) ];
   9: [XIO(LN98_Break_LineWide) MOV(LN98_TO_DC1_MAIN_MESSAGE_A[3],LN98NAM02) ,XIC(LN98_Break_LineWide) MOV(0,LN98NAM02) ];
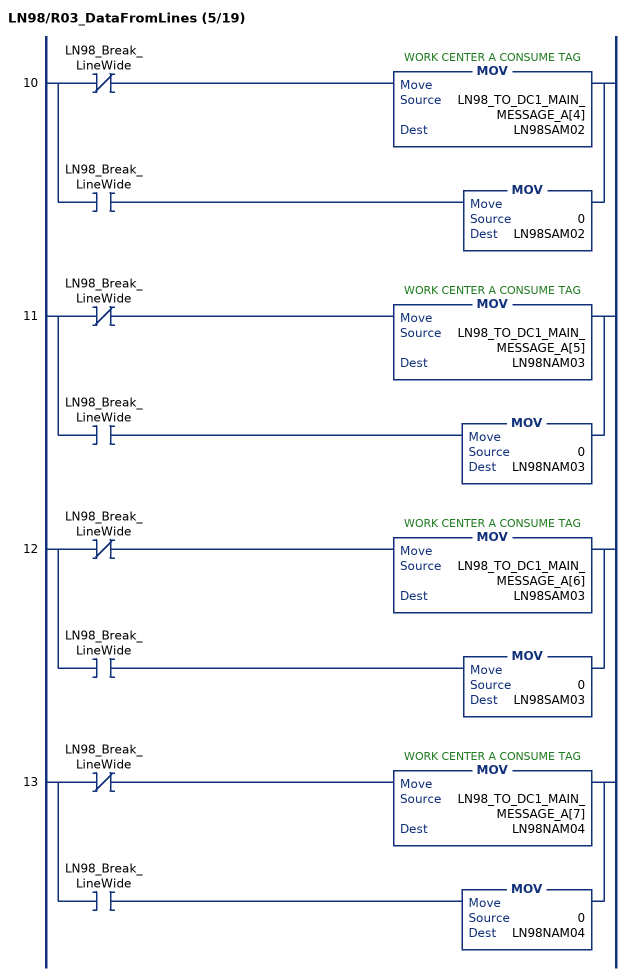
   10: [XIO(LN98_Break_LineWide) MOV(LN98_TO_DC1_MAIN_MESSAGE_A[4],LN98SAM02) ,XIC(LN98_Break_LineWide) MOV(0,LN98SAM02) ];
   11: [XIO(LN98_Break_LineWide) MOV(LN98_TO_DC1_MAIN_MESSAGE_A[5],LN98NAM03) ,XIC(LN98_Break_LineWide) MOV(0,LN98NAM03) ];
   12: [XIO(LN98_Break_LineWide) MOV(LN98_TO_DC1_MAIN_MESSAGE_A[6],LN98SAM03) ,XIC(LN98_Break_LineWide) MOV(0,LN98SAM03) ];
   13: [XIO(LN98_Break_LineWide) MOV(LN98_TO_DC1_MAIN_MESSAGE_A[7],LN98NAM04) ,XIC(LN98_Break_LineWide) MOV(0,LN98NAM04) ];
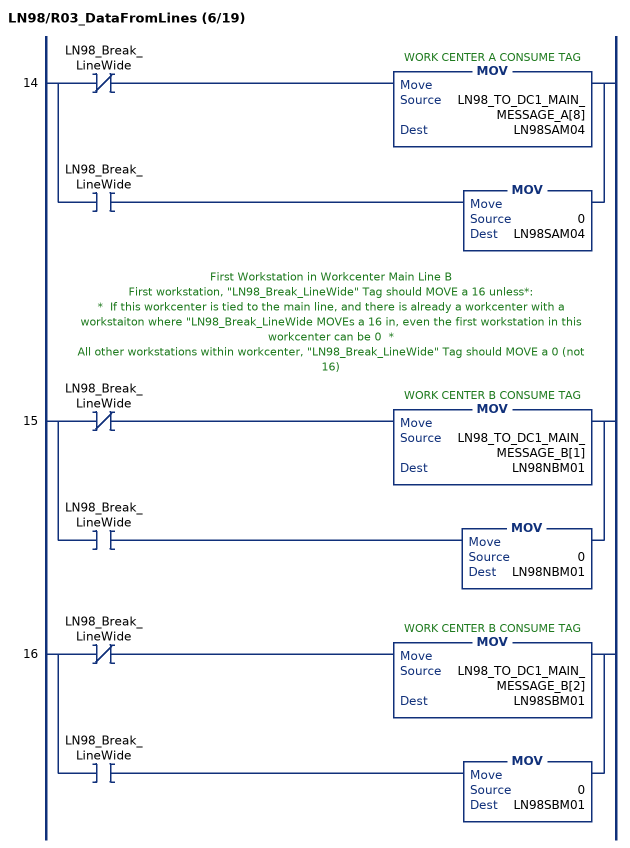
   14: [XIO(LN98_Break_LineWide) MOV(LN98_TO_DC1_MAIN_MESSAGE_A[8],LN98SAM04) ,XIC(LN98_Break_LineWide) MOV(0,LN98SAM04) ];
   // First Workstation in Workcenter Main Line B
   // First workstation, "LN98_Break_LineWide" Tag should MOVE a 16 unless*:
   // *  If this workcenter is tied to the main line, and there is already a workcenter with a workstaiton where "LN98_Break_LineWide MOVEs a 16 in, even the first workstation in this workcenter can be 0  *
   // All other workstations within workcenter, "LN98_Break_LineWide" Tag should MOVE a 0 (not 16)
   15: [XIO(LN98_Break_LineWide) MOV(LN98_TO_DC1_MAIN_MESSAGE_B[1],LN98NBM01) ,XIC(LN98_Break_LineWide) MOV(0,LN98NBM01) ];
   16: [XIO(LN98_Break_LineWide) MOV(LN98_TO_DC1_MAIN_MESSAGE_B[2],LN98SBM01) ,XIC(LN98_Break_LineWide) MOV(0,LN98SBM01) ];
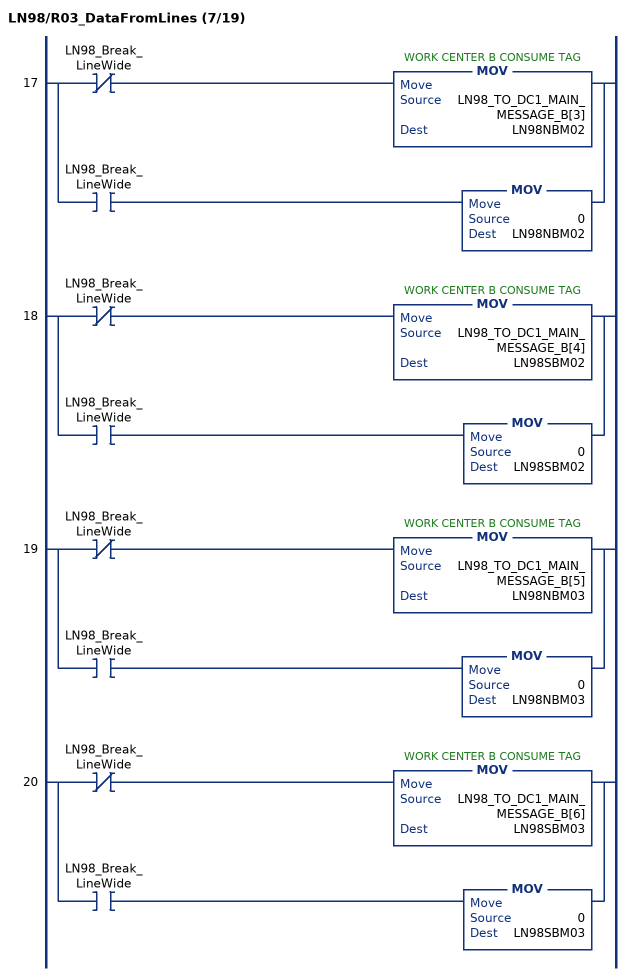
   17: [XIO(LN98_Break_LineWide) MOV(LN98_TO_DC1_MAIN_MESSAGE_B[3],LN98NBM02) ,XIC(LN98_Break_LineWide) MOV(0,LN98NBM02) ];
   18: [XIO(LN98_Break_LineWide) MOV(LN98_TO_DC1_MAIN_MESSAGE_B[4],LN98SBM02) ,XIC(LN98_Break_LineWide) MOV(0,LN98SBM02) ];
   19: [XIO(LN98_Break_LineWide) MOV(LN98_TO_DC1_MAIN_MESSAGE_B[5],LN98NBM03) ,XIC(LN98_Break_LineWide) MOV(0,LN98NBM03) ];
   20: [XIO(LN98_Break_LineWide) MOV(LN98_TO_DC1_MAIN_MESSAGE_B[6],LN98SBM03) ,XIC(LN98_Break_LineWide) MOV(0,LN98SBM03) ];
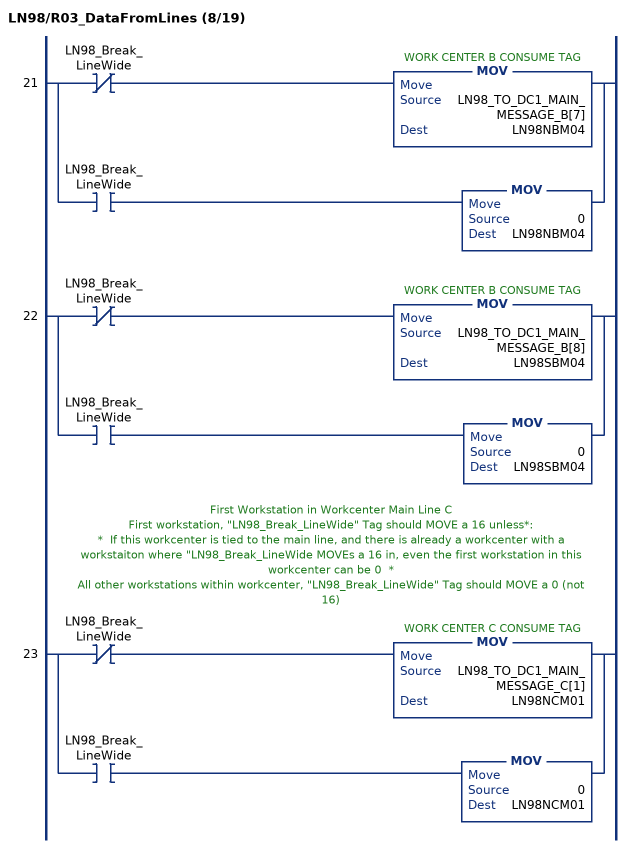
   21: [XIO(LN98_Break_LineWide) MOV(LN98_TO_DC1_MAIN_MESSAGE_B[7],LN98NBM04) ,XIC(LN98_Break_LineWide) MOV(0,LN98NBM04) ];
   22: [XIO(LN98_Break_LineWide) MOV(LN98_TO_DC1_MAIN_MESSAGE_B[8],LN98SBM04) ,XIC(LN98_Break_LineWide) MOV(0,LN98SBM04) ];
   // First Workstation in Workcenter Main Line C
   // First workstation, "LN98_Break_LineWide" Tag should MOVE a 16 unless*:
   // *  If this workcenter is tied to the main line, and there is already a workcenter with a workstaiton where "LN98_Break_LineWide MOVEs a 16 in, even the first workstation in this workcenter can be 0  *
   // All other workstations within workcenter, "LN98_Break_LineWide" Tag should MOVE a 0 (not 16)
   23: [XIO(LN98_Break_LineWide) MOV(LN98_TO_DC1_MAIN_MESSAGE_C[1],LN98NCM01) ,XIC(LN98_Break_LineWide) MOV(0,LN98NCM01) ];
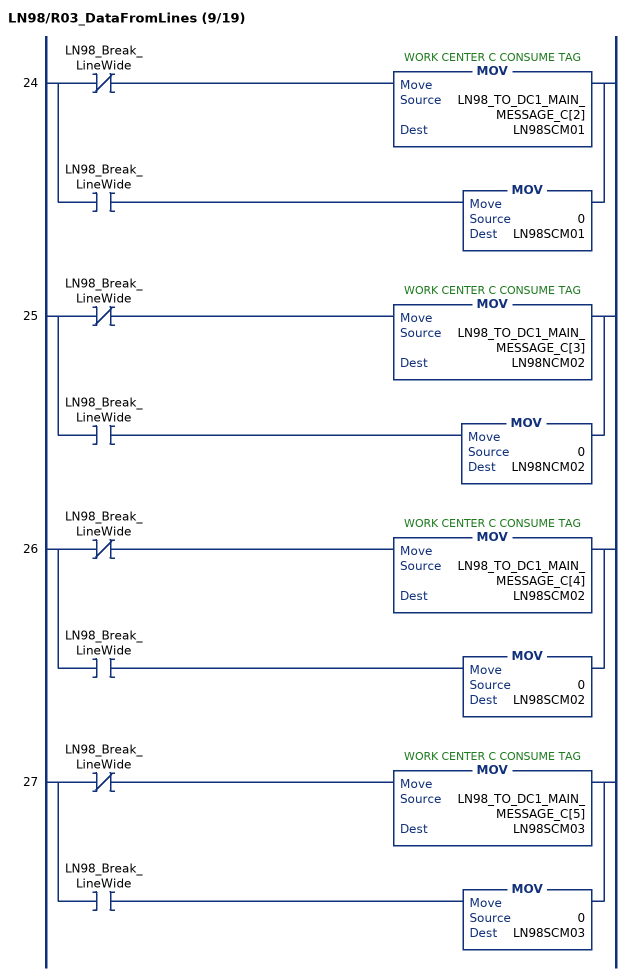
   24: [XIO(LN98_Break_LineWide) MOV(LN98_TO_DC1_MAIN_MESSAGE_C[2],LN98SCM01) ,XIC(LN98_Break_LineWide) MOV(0,LN98SCM01) ];
   25: [XIO(LN98_Break_LineWide) MOV(LN98_TO_DC1_MAIN_MESSAGE_C[3],LN98NCM02) ,XIC(LN98_Break_LineWide) MOV(0,LN98NCM02) ];
   26: [XIO(LN98_Break_LineWide) MOV(LN98_TO_DC1_MAIN_MESSAGE_C[4],LN98SCM02) ,XIC(LN98_Break_LineWide) MOV(0,LN98SCM02) ];
   27: [XIO(LN98_Break_LineWide) MOV(LN98_TO_DC1_MAIN_MESSAGE_C[5],LN98SCM03) ,XIC(LN98_Break_LineWide) MOV(0,LN98SCM03) ];
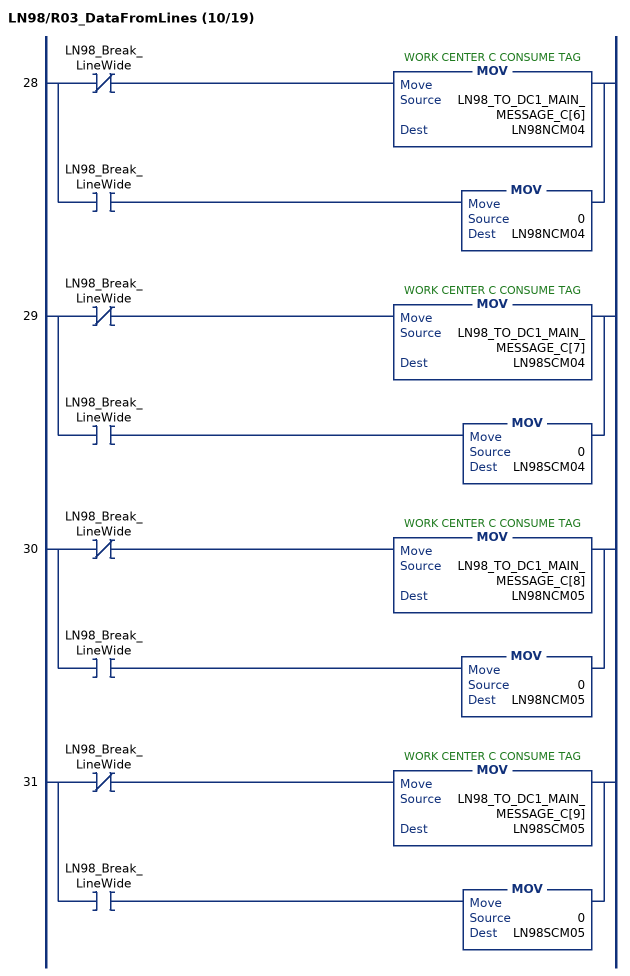
   28: [XIO(LN98_Break_LineWide) MOV(LN98_TO_DC1_MAIN_MESSAGE_C[6],LN98NCM04) ,XIC(LN98_Break_LineWide) MOV(0,LN98NCM04) ];
   29: [XIO(LN98_Break_LineWide) MOV(LN98_TO_DC1_MAIN_MESSAGE_C[7],LN98SCM04) ,XIC(LN98_Break_LineWide) MOV(0,LN98SCM04) ];
   30: [XIO(LN98_Break_LineWide) MOV(LN98_TO_DC1_MAIN_MESSAGE_C[8],LN98NCM05) ,XIC(LN98_Break_LineWide) MOV(0,LN98NCM05) ];
   31: [XIO(LN98_Break_LineWide) MOV(LN98_TO_DC1_MAIN_MESSAGE_C[9],LN98SCM05) ,XIC(LN98_Break_LineWide) MOV(0,LN98SCM05) ];
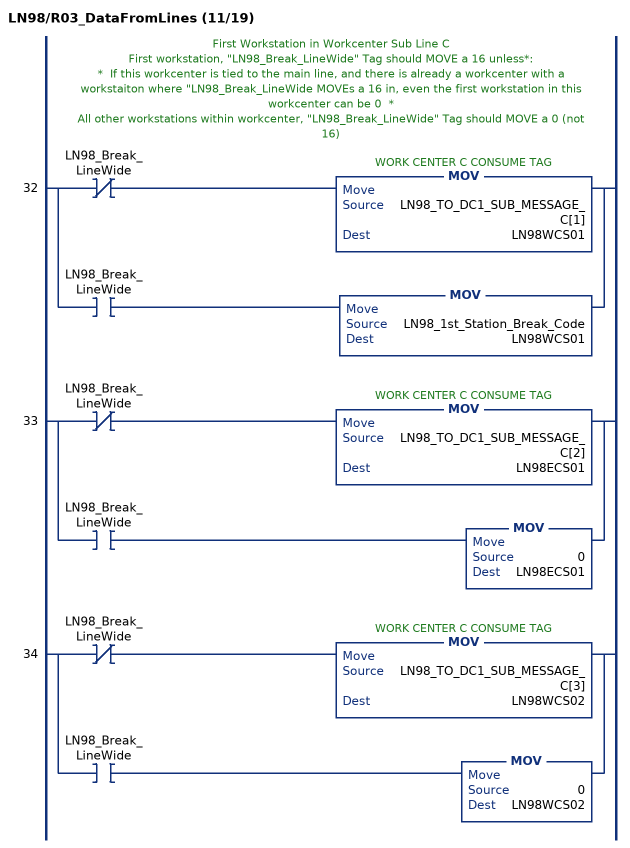
   // First Workstation in Workcenter Sub Line C
   // First workstation, "LN98_Break_LineWide" Tag should MOVE a 16 unless*:
   // *  If this workcenter is tied to the main line, and there is already a workcenter with a workstaiton where "LN98_Break_LineWide MOVEs a 16 in, even the first workstation in this workcenter can be 0  *
   // All other workstations within workcenter, "LN98_Break_LineWide" Tag should MOVE a 0 (not 16)
   32: [XIO(LN98_Break_LineWide) MOV(LN98_TO_DC1_SUB_MESSAGE_C[1],LN98WCS01) ,XIC(LN98_Break_LineWide) MOV(LN98_1st_Station_Break_Code,LN98WCS01) ];
   33: [XIO(LN98_Break_LineWide) MOV(LN98_TO_DC1_SUB_MESSAGE_C[2],LN98ECS01) ,XIC(LN98_Break_LineWide) MOV(0,LN98ECS01) ];
   34: [XIO(LN98_Break_LineWide) MOV(LN98_TO_DC1_SUB_MESSAGE_C[3],LN98WCS02) ,XIC(LN98_Break_LineWide) MOV(0,LN98WCS02) ];
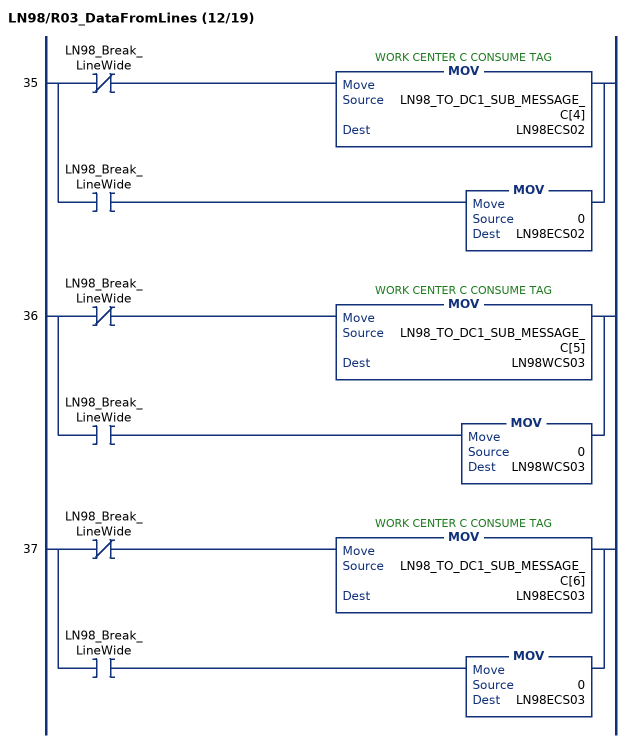
   35: [XIO(LN98_Break_LineWide) MOV(LN98_TO_DC1_SUB_MESSAGE_C[4],LN98ECS02) ,XIC(LN98_Break_LineWide) MOV(0,LN98ECS02) ];
   36: [XIO(LN98_Break_LineWide) MOV(LN98_TO_DC1_SUB_MESSAGE_C[5],LN98WCS03) ,XIC(LN98_Break_LineWide) MOV(0,LN98WCS03) ];
   37: [XIO(LN98_Break_LineWide) MOV(LN98_TO_DC1_SUB_MESSAGE_C[6],LN98ECS03) ,XIC(LN98_Break_LineWide) MOV(0,LN98ECS03) ];
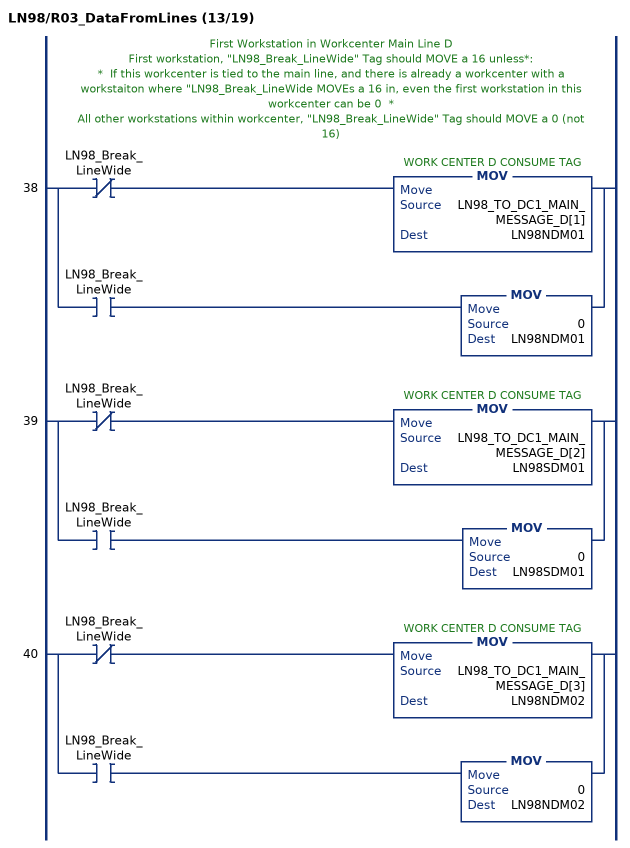
   // First Workstation in Workcenter Main Line D
   // First workstation, "LN98_Break_LineWide" Tag should MOVE a 16 unless*:
   // *  If this workcenter is tied to the main line, and there is already a workcenter with a workstaiton where "LN98_Break_LineWide MOVEs a 16 in, even the first workstation in this workcenter can be 0  *
   // All other workstations within workcenter, "LN98_Break_LineWide" Tag should MOVE a 0 (not 16)
   38: [XIO(LN98_Break_LineWide) MOV(LN98_TO_DC1_MAIN_MESSAGE_D[1],LN98NDM01) ,XIC(LN98_Break_LineWide) MOV(0,LN98NDM01) ];
   39: [XIO(LN98_Break_LineWide) MOV(LN98_TO_DC1_MAIN_MESSAGE_D[2],LN98SDM01) ,XIC(LN98_Break_LineWide) MOV(0,LN98SDM01) ];
   40: [XIO(LN98_Break_LineWide) MOV(LN98_TO_DC1_MAIN_MESSAGE_D[3],LN98NDM02) ,XIC(LN98_Break_LineWide) MOV(0,LN98NDM02) ];
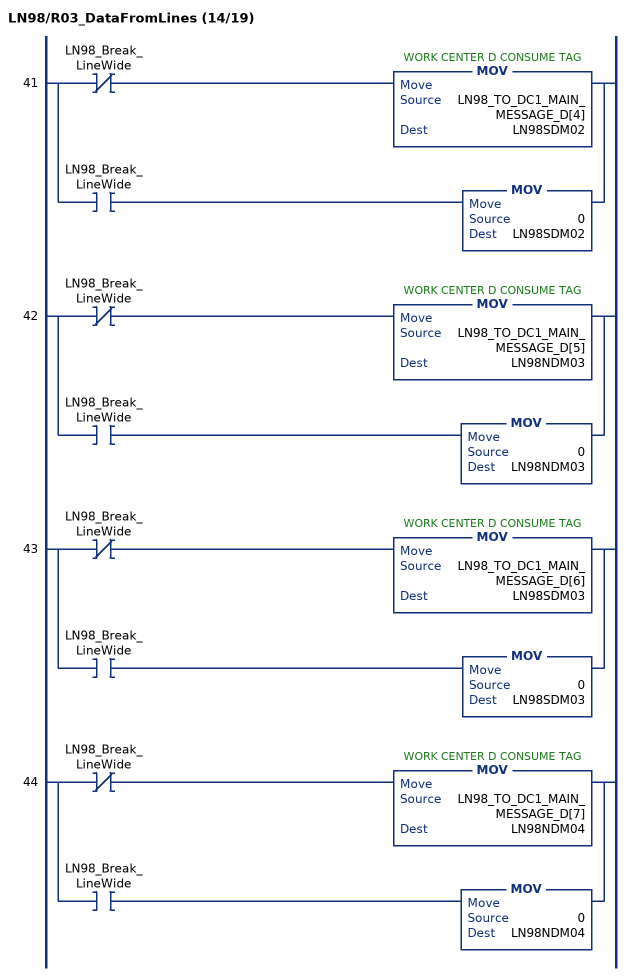
   41: [XIO(LN98_Break_LineWide) MOV(LN98_TO_DC1_MAIN_MESSAGE_D[4],LN98SDM02) ,XIC(LN98_Break_LineWide) MOV(0,LN98SDM02) ];
   42: [XIO(LN98_Break_LineWide) MOV(LN98_TO_DC1_MAIN_MESSAGE_D[5],LN98NDM03) ,XIC(LN98_Break_LineWide) MOV(0,LN98NDM03) ];
   43: [XIO(LN98_Break_LineWide) MOV(LN98_TO_DC1_MAIN_MESSAGE_D[6],LN98SDM03) ,XIC(LN98_Break_LineWide) MOV(0,LN98SDM03) ];
   44: [XIO(LN98_Break_LineWide) MOV(LN98_TO_DC1_MAIN_MESSAGE_D[7],LN98NDM04) ,XIC(LN98_Break_LineWide) MOV(0,LN98NDM04) ];
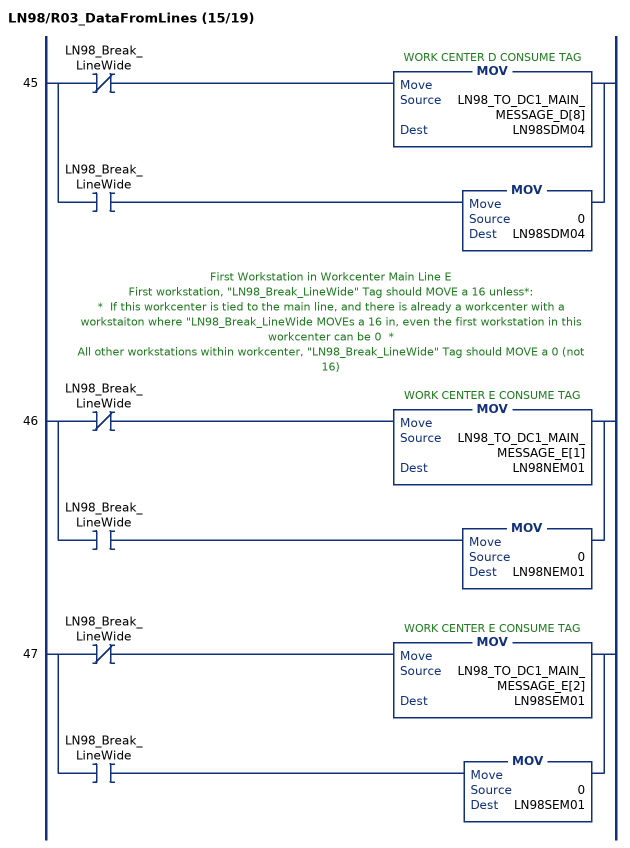
   45: [XIO(LN98_Break_LineWide) MOV(LN98_TO_DC1_MAIN_MESSAGE_D[8],LN98SDM04) ,XIC(LN98_Break_LineWide) MOV(0,LN98SDM04) ];
   // First Workstation in Workcenter Main Line E
   // First workstation, "LN98_Break_LineWide" Tag should MOVE a 16 unless*:
   // *  If this workcenter is tied to the main line, and there is already a workcenter with a workstaiton where "LN98_Break_LineWide MOVEs a 16 in, even the first workstation in this workcenter can be 0  *
   // All other workstations within workcenter, "LN98_Break_LineWide" Tag should MOVE a 0 (not 16)
   46: [XIO(LN98_Break_LineWide) MOV(LN98_TO_DC1_MAIN_MESSAGE_E[1],LN98NEM01) ,XIC(LN98_Break_LineWide) MOV(0,LN98NEM01) ];
   47: [XIO(LN98_Break_LineWide) MOV(LN98_TO_DC1_MAIN_MESSAGE_E[2],LN98SEM01) ,XIC(LN98_Break_LineWide) MOV(0,LN98SEM01) ];
